Yaskawa INFORM job: test_long_tjr0.JBI

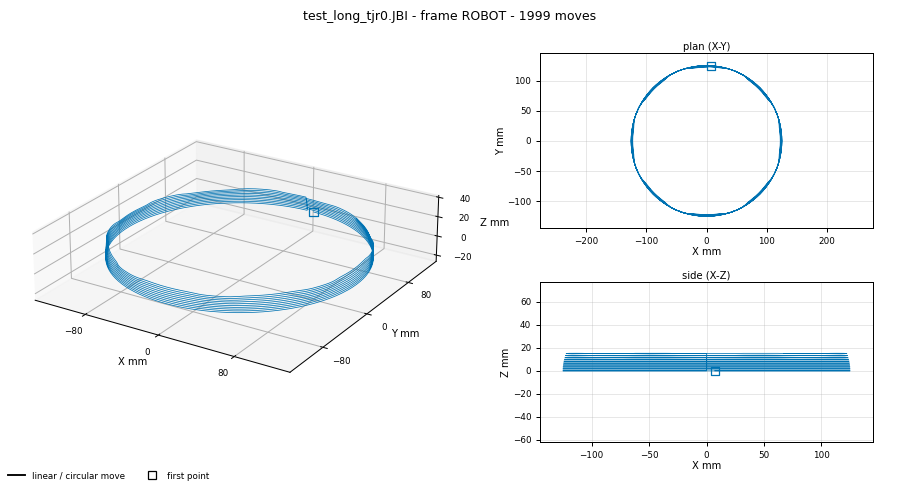
[picture p0: tool path of test_long_tjr0.JBI in frame ROBOT, 1999 of 2000 moves have a stored position in this frame; points joined in program order, loops and branches not executed]
version: 0
/JOB
//NAME test_long
//POS
///NPOS 48,0,0,2,0,0
///TOOL 1
///POSTYPE ROBOT
///RECTAN
///RCONF 1,0,0,0,0,0,0,0,0,0,0,0,0,0,0,0,0,0,0,0,0,0,0,0
C00000=0.000,125.000,0.000,0.0000,0.0000,1.0000
C00001=7.240,124.790,0.000,-0.0000,0.0000,1.0000
C00002=13.740,124.240,0.000,-0.0000,0.0000,1.0000
C00003=19.450,123.480,0.000,-0.0000,0.0000,1.0000
C00004=23.370,122.800,0.000,-0.0000,0.0000,1.0000
C00005=26.070,122.250,0.000,-0.0000,0.0000,1.0000
C00006=28.240,121.770,0.000,-0.0000,-0.0000,1.0000
C00007=30.440,121.240,0.000,-0.0000,-0.0000,1.0000
C00008=33.190,120.510,0.000,-0.0000,0.0000,1.0000
C00009=36.560,119.530,0.000,-0.0000,0.0000,1.0000
C00010=40.120,118.390,0.000,-0.0000,0.0000,1.0000
C00011=43.420,117.220,0.000,-0.0000,0.0000,1.0000
C00012=46.400,116.070,0.000,-0.0000,0.0000,1.0000
C00013=49.260,114.880,0.000,-0.0000,0.0000,1.0000
C00014=52.180,113.590,0.000,-0.0000,0.0000,1.0000
C00015=55.350,112.080,0.000,0.0000,0.0000,1.0000
C00016=58.670,110.370,0.000,0.0000,0.0000,1.0000
C00017=61.750,108.680,0.000,-0.0000,0.0000,1.0000
C00018=64.200,107.250,0.000,-0.0000,0.0000,1.0000
C00019=66.130,106.070,0.000,-0.0000,0.0000,1.0000
C00020=68.010,104.880,0.000,-0.0000,0.0000,1.0000
C00021=70.300,103.360,0.000,-0.0000,0.0000,1.0000
C00022=73.550,101.070,0.000,-0.0000,0.0000,1.0000
C00023=78.140,97.570,0.000,-0.0000,0.0000,1.0000
C00024=83.120,93.360,0.000,-0.0000,0.0000,1.0000
C00025=88.390,88.390,0.000,-0.0000,0.0000,1.0000
C00026=93.360,83.120,0.000,-0.0000,0.0000,1.0000
C00027=97.570,78.140,0.000,-0.0000,0.0000,1.0000
C00028=101.070,73.550,0.000,0.0000,0.0000,1.0000
C00029=103.360,70.300,0.000,-0.0000,0.0000,1.0000
C00030=104.880,68.010,0.000,-0.0000,0.0000,1.0000
C00031=106.070,66.130,0.000,-0.0000,0.0000,1.0000
C00032=107.250,64.200,0.000,-0.0000,0.0000,1.0000
C00033=108.680,61.750,0.000,-0.0000,0.0000,1.0000
C00034=110.370,58.670,0.000,-0.0000,0.0000,1.0000
C00035=112.080,55.350,0.000,-0.0000,0.0000,1.0000
C00036=113.590,52.180,0.000,-0.0000,0.0000,1.0000
C00037=114.880,49.260,0.000,-0.0000,0.0000,1.0000
C00038=116.070,46.400,0.000,-0.0000,0.0000,1.0000
C00039=117.220,43.420,0.000,-0.0000,0.0000,1.0000
C00040=118.390,40.120,0.000,-0.0000,0.0000,1.0000
C00041=119.530,36.560,0.000,-0.0000,0.0000,1.0000
C00042=120.510,33.190,0.000,-0.0000,0.0000,1.0000
C00043=121.240,30.440,0.000,-0.0000,0.0000,1.0000
C00044=121.770,28.240,0.000,-0.0000,0.0000,1.0000
C00045=122.250,26.070,0.000,-0.0000,0.0000,1.0000
C00046=122.800,23.370,0.000,-0.0000,0.0000,1.0000
C00047=123.480,19.450,0.000,-0.0000,0.0000,1.0000
C00048=124.240,13.740,0.000,-0.0000,0.0000,1.0000
C00049=124.790,7.240,0.000,-0.0000,0.0000,1.0000
C00050=125.000,0.000,0.000,-0.0000,0.0000,1.0000
C00051=124.790,-7.240,0.000,0.0000,0.0000,1.0000
C00052=124.240,-13.740,0.000,0.0000,0.0000,1.0000
C00053=123.480,-19.450,0.000,0.0000,0.0000,1.0000
C00054=122.800,-23.370,0.000,0.0000,0.0000,1.0000
C00055=122.250,-26.070,0.000,0.0000,0.0000,1.0000
C00056=121.770,-28.240,0.000,-0.0000,0.0000,1.0000
C00057=121.240,-30.440,0.000,-0.0000,0.0000,1.0000
C00058=120.510,-33.190,0.000,0.0000,0.0000,1.0000
C00059=119.530,-36.560,0.000,0.0000,0.0000,1.0000
C00060=118.390,-40.120,0.000,0.0000,0.0000,1.0000
C00061=117.220,-43.420,0.000,0.0000,0.0000,1.0000
C00062=116.070,-46.400,0.000,0.0000,0.0000,1.0000
C00063=114.880,-49.260,0.000,0.0000,0.0000,1.0000
C00064=113.590,-52.180,0.000,0.0000,0.0000,1.0000
C00065=112.080,-55.350,0.000,0.0000,0.0000,1.0000
C00066=110.370,-58.670,0.000,0.0000,0.0000,1.0000
C00067=108.680,-61.750,0.000,0.0000,0.0000,1.0000
C00068=107.250,-64.200,0.000,0.0000,0.0000,1.0000
C00069=106.070,-66.130,0.000,0.0000,0.0000,1.0000
C00070=104.880,-68.010,0.000,0.0000,0.0000,1.0000
C00071=103.360,-70.300,0.000,0.0000,0.0000,1.0000
C00072=101.070,-73.550,0.000,0.0000,0.0000,1.0000
C00073=97.570,-78.140,0.000,0.0000,0.0000,1.0000
C00074=93.360,-83.120,0.000,0.0000,0.0000,1.0000
C00075=88.390,-88.390,0.000,0.0000,0.0000,1.0000
C00076=83.120,-93.360,0.000,0.0000,0.0000,1.0000
C00077=78.140,-97.570,0.000,0.0000,0.0000,1.0000
C00078=73.550,-101.070,0.000,0.0000,0.0000,1.0000
C00079=70.300,-103.360,0.000,0.0000,0.0000,1.0000
C00080=68.010,-104.880,0.000,0.0000,0.0000,1.0000
C00081=66.130,-106.070,0.000,0.0000,0.0000,1.0000
C00082=64.200,-107.250,0.000,0.0000,0.0000,1.0000
C00083=61.750,-108.680,0.000,0.0000,-0.0000,1.0000
C00084=58.670,-110.370,0.000,0.0000,0.0000,1.0000
C00085=55.350,-112.080,0.000,0.0000,0.0000,1.0000
C00086=52.180,-113.590,0.000,0.0000,0.0000,1.0000
C00087=49.260,-114.880,0.000,0.0000,0.0000,1.0000
C00088=46.400,-116.070,0.000,0.0000,0.0000,1.0000
C00089=43.420,-117.220,0.000,0.0000,0.0000,1.0000
C00090=40.120,-118.390,0.000,0.0000,0.0000,1.0000
C00091=36.560,-119.530,0.000,0.0000,0.0000,1.0000
C00092=33.190,-120.510,0.000,0.0000,0.0000,1.0000
C00093=30.440,-121.240,0.000,0.0000,0.0000,1.0000
C00094=28.240,-121.770,0.000,0.0000,0.0000,1.0000
C00095=26.070,-122.250,0.000,0.0000,0.0000,1.0000
C00096=23.370,-122.800,0.000,0.0000,0.0000,1.0000
C00097=19.450,-123.480,0.000,0.0000,0.0000,1.0000
C00098=13.740,-124.240,0.000,0.0000,0.0000,1.0000
C00099=7.240,-124.790,0.000,0.0000,0.0000,1.0000
C00100=0.000,-125.000,0.000,0.0000,-0.0000,1.0000
C00101=0.000,-125.000,0.000,0.0000,-0.0000,1.0000
C00102=-7.240,-124.790,0.000,0.0000,-0.0000,1.0000
C00103=-13.740,-124.240,0.000,0.0000,-0.0000,1.0000
C00104=-19.450,-123.480,0.000,0.0000,-0.0000,1.0000
C00105=-23.370,-122.800,0.000,-0.0000,-0.0000,1.0000
C00106=-26.070,-122.250,0.000,0.0000,-0.0000,1.0000
C00107=-28.240,-121.770,0.000,0.0000,-0.0000,1.0000
C00108=-30.440,-121.240,0.000,0.0000,-0.0000,1.0000
C00109=-33.190,-120.510,0.000,0.0000,-0.0000,1.0000
C00110=-36.560,-119.530,0.000,0.0000,-0.0000,1.0000
C00111=-40.120,-118.390,0.000,0.0000,-0.0000,1.0000
C00112=-43.420,-117.220,0.000,0.0000,-0.0000,1.0000
C00113=-46.400,-116.070,0.000,0.0000,-0.0000,1.0000
C00114=-49.260,-114.880,0.000,0.0000,-0.0000,1.0000
C00115=-52.180,-113.590,0.000,0.0000,-0.0000,1.0000
C00116=-55.350,-112.080,0.000,0.0000,-0.0000,1.0000
C00117=-58.670,-110.370,0.000,0.0000,-0.0000,1.0000
C00118=-61.750,-108.680,0.000,0.0000,-0.0000,1.0000
C00119=-64.200,-107.250,0.000,0.0000,-0.0000,1.0000
C00120=-66.130,-106.070,0.000,0.0000,-0.0000,1.0000
C00121=-68.010,-104.880,0.000,0.0000,-0.0000,1.0000
C00122=-70.300,-103.360,0.000,0.0000,-0.0000,1.0000
C00123=-73.550,-101.070,0.000,0.0000,-0.0000,1.0000
C00124=-78.140,-97.570,0.000,0.0000,-0.0000,1.0000
C00125=-83.120,-93.360,0.000,0.0000,-0.0000,1.0000
C00126=-88.390,-88.390,0.000,0.0000,-0.0000,1.0000
C00127=-93.360,-83.120,0.000,0.0000,-0.0000,1.0000
C00128=-97.570,-78.140,0.000,0.0000,-0.0000,1.0000
C00129=-101.070,-73.550,0.000,0.0000,-0.0000,1.0000
C00130=-103.360,-70.300,0.000,0.0000,-0.0000,1.0000
C00131=-104.880,-68.010,0.000,0.0000,-0.0000,1.0000
C00132=-106.070,-66.130,0.000,0.0000,-0.0000,1.0000
C00133=-107.250,-64.200,0.000,0.0000,-0.0000,1.0000
C00134=-108.680,-61.750,0.000,0.0000,-0.0000,1.0000
C00135=-110.370,-58.670,0.000,0.0000,-0.0000,1.0000
C00136=-112.080,-55.350,0.000,0.0000,-0.0000,1.0000
C00137=-113.590,-52.180,0.000,0.0000,0.0000,1.0000
C00138=-114.880,-49.260,0.000,0.0000,0.0000,1.0000
C00139=-116.070,-46.400,0.000,0.0000,-0.0000,1.0000
C00140=-117.220,-43.420,0.000,0.0000,-0.0000,1.0000
C00141=-118.390,-40.120,0.000,0.0000,0.0000,1.0000
C00142=-119.530,-36.560,0.000,0.0000,0.0000,1.0000
C00143=-120.510,-33.190,0.000,0.0000,-0.0000,1.0000
C00144=-121.240,-30.440,0.000,0.0000,-0.0000,1.0000
C00145=-121.770,-28.240,0.000,0.0000,-0.0000,1.0000
C00146=-122.250,-26.070,0.000,0.0000,-0.0000,1.0000
C00147=-122.800,-23.370,0.000,0.0000,-0.0000,1.0000
C00148=-123.480,-19.450,0.000,0.0000,-0.0000,1.0000
C00149=-124.240,-13.740,0.000,0.0000,-0.0000,1.0000
C00150=-124.790,-7.240,0.000,0.0000,-0.0000,1.0000
C00151=-125.000,0.000,0.000,0.0000,0.0000,1.0000
C00152=-124.790,7.240,0.000,0.0000,0.0000,1.0000
C00153=-124.240,13.740,0.000,0.0000,0.0000,1.0000
C00154=-123.480,19.450,0.000,0.0000,0.0000,1.0000
C00155=-122.800,23.370,0.000,0.0000,0.0000,1.0000
C00156=-122.250,26.070,0.000,0.0000,0.0000,1.0000
C00157=-121.770,28.240,0.000,0.0000,0.0000,1.0000
C00158=-121.240,30.440,0.000,0.0000,0.0000,1.0000
C00159=-120.510,33.190,0.000,0.0000,0.0000,1.0000
C00160=-119.530,36.560,0.000,0.0000,0.0000,1.0000
C00161=-118.390,40.120,0.000,0.0000,0.0000,1.0000
C00162=-117.220,43.420,0.000,0.0000,0.0000,1.0000
C00163=-116.070,46.400,0.000,0.0000,0.0000,1.0000
C00164=-114.880,49.260,0.000,0.0000,0.0000,1.0000
C00165=-113.590,52.180,0.000,0.0000,0.0000,1.0000
C00166=-112.080,55.350,0.000,0.0000,0.0000,1.0000
C00167=-110.370,58.670,0.000,0.0000,0.0000,1.0000
C00168=-108.680,61.750,0.000,0.0000,0.0000,1.0000
C00169=-107.250,64.200,0.000,0.0000,0.0000,1.0000
C00170=-106.070,66.130,0.000,0.0000,0.0000,1.0000
C00171=-104.880,68.010,0.000,0.0000,0.0000,1.0000
C00172=-103.360,70.300,0.000,0.0000,0.0000,1.0000
C00173=-101.070,73.550,0.000,0.0000,0.0000,1.0000
C00174=-97.570,78.140,0.000,0.0000,0.0000,1.0000
C00175=-93.360,83.120,0.000,0.0000,0.0000,1.0000
C00176=-88.390,88.390,0.000,0.0000,0.0000,1.0000
C00177=-83.120,93.360,0.000,0.0000,0.0000,1.0000
C00178=-78.140,97.570,0.000,0.0000,0.0000,1.0000
C00179=-73.550,101.070,0.000,0.0000,0.0000,1.0000
C00180=-70.300,103.360,0.000,0.0000,0.0000,1.0000
C00181=-68.010,104.880,0.000,0.0000,0.0000,1.0000
C00182=-66.130,106.070,0.000,0.0000,0.0000,1.0000
C00183=-64.200,107.250,0.000,0.0000,0.0000,1.0000
C00184=-61.750,108.680,0.000,0.0000,0.0000,1.0000
C00185=-58.670,110.370,0.000,0.0000,0.0000,1.0000
C00186=-55.350,112.080,0.000,0.0000,0.0000,1.0000
C00187=-52.180,113.590,0.000,0.0000,0.0000,1.0000
C00188=-49.260,114.880,0.000,0.0000,0.0000,1.0000
C00189=-46.400,116.070,0.000,0.0000,0.0000,1.0000
C00190=-43.420,117.220,0.000,0.0000,0.0000,1.0000
C00191=-40.120,118.390,0.000,0.0000,-0.0000,1.0000
C00192=-36.560,119.530,0.000,0.0000,-0.0000,1.0000
C00193=-33.190,120.510,0.000,0.0000,0.0000,1.0000
C00194=-30.440,121.240,0.000,0.0000,0.0000,1.0000
C00195=-28.240,121.770,0.000,0.0000,0.0000,1.0000
C00196=-26.070,122.250,0.000,0.0000,0.0000,1.0000
C00197=-23.370,122.800,0.000,0.0000,0.0000,1.0000
C00198=-19.450,123.480,0.000,0.0000,0.0000,1.0000
C00199=-13.740,124.240,0.000,0.0000,0.0000,1.0000
C00200=-7.240,124.790,0.000,0.0000,0.0000,1.0000
C00201=0.000,125.000,0.000,0.0000,0.0000,1.0000
C00202=0.000,124.960,1.700,0.0000,-0.0400,1.0000
C00203=-7.240,124.750,1.700,0.0000,-0.0400,1.0000
C00204=-13.730,124.210,1.700,0.0000,-0.0400,1.0000
C00205=-19.450,123.440,1.700,0.0100,-0.0400,1.0000
C00206=-23.360,122.760,1.700,0.0100,-0.0400,1.0000
C00207=-26.060,122.230,1.700,0.0100,-0.0300,1.0000
C00208=-28.230,121.750,1.700,0.0100,-0.0200,1.0000
C00209=-30.430,121.230,1.700,0.0000,-0.0200,1.0000
C00210=-33.180,120.510,1.700,0.0000,-0.0100,1.0000
C00211=-36.550,119.530,1.700,0.0000,-0.0000,1.0000
C00212=-40.110,118.390,1.700,0.0000,-0.0000,1.0000
C00213=-43.420,117.220,1.700,0.0000,-0.0000,1.0000
C00214=-46.400,116.070,1.700,0.0000,-0.0000,1.0000
C00215=-49.260,114.880,1.700,0.0000,-0.0000,1.0000
C00216=-52.180,113.590,1.700,0.0000,-0.0000,1.0000
C00217=-55.350,112.080,1.700,0.0000,-0.0000,1.0000
C00218=-58.680,110.370,1.700,0.0000,-0.0000,1.0000
C00219=-61.750,108.670,1.700,0.0100,-0.0100,1.0000
C00220=-64.200,107.240,1.700,0.0100,-0.0100,1.0000
C00221=-66.130,106.050,1.700,0.0100,-0.0200,1.0000
C00222=-68.000,104.850,1.700,0.0200,-0.0300,1.0000
C00223=-70.290,103.330,1.700,0.0200,-0.0300,1.0000
C00224=-73.530,101.040,1.700,0.0300,-0.0300,1.0000
C00225=-78.120,97.540,1.700,0.0300,-0.0300,1.0000
C00226=-83.100,93.330,1.700,0.0300,-0.0300,1.0000
C00227=-88.360,88.360,1.700,0.0300,-0.0300,1.0000
C00228=-93.330,83.100,1.700,0.0300,-0.0300,1.0000
C00229=-97.540,78.120,1.700,0.0300,-0.0300,1.0000
C00230=-101.040,73.530,1.700,0.0300,-0.0300,1.0000
C00231=-103.330,70.290,1.700,0.0300,-0.0200,1.0000
C00232=-104.850,68.000,1.700,0.0300,-0.0200,1.0000
C00233=-106.050,66.130,1.700,0.0200,-0.0100,1.0000
C00234=-107.240,64.200,1.700,0.0100,-0.0100,1.0000
C00235=-108.670,61.750,1.700,0.0100,-0.0100,1.0000
C00236=-110.370,58.680,1.700,0.0000,-0.0000,1.0000
C00237=-112.080,55.350,1.700,0.0000,-0.0000,1.0000
C00238=-113.590,52.180,1.700,0.0000,-0.0000,1.0000
C00239=-114.880,49.260,1.700,0.0000,-0.0000,1.0000
C00240=-116.070,46.400,1.700,0.0000,-0.0000,1.0000
C00241=-117.220,43.420,1.700,0.0000,-0.0000,1.0000
C00242=-118.390,40.110,1.700,0.0000,-0.0000,1.0000
C00243=-119.530,36.550,1.700,0.0000,-0.0000,1.0000
C00244=-120.510,33.180,1.700,0.0100,-0.0000,1.0000
C00245=-121.230,30.430,1.700,0.0200,-0.0000,1.0000
C00246=-121.750,28.230,1.700,0.0200,-0.0100,1.0000
C00247=-122.230,26.060,1.700,0.0300,-0.0100,1.0000
C00248=-122.760,23.360,1.700,0.0400,-0.0100,1.0000
C00249=-123.440,19.450,1.700,0.0400,-0.0100,1.0000
C00250=-124.210,13.730,1.700,0.0400,-0.0000,1.0000
C00251=-124.750,7.240,1.700,0.0400,-0.0000,1.0000
C00252=-124.960,0.000,1.700,0.0400,-0.0000,1.0000
C00253=-124.750,-7.240,1.700,0.0400,0.0000,1.0000
C00254=-124.210,-13.730,1.700,0.0400,0.0000,1.0000
C00255=-123.440,-19.450,1.700,0.0400,0.0100,1.0000
C00256=-122.760,-23.360,1.700,0.0400,0.0100,1.0000
C00257=-122.230,-26.060,1.700,0.0300,0.0100,1.0000
C00258=-121.750,-28.230,1.700,0.0200,0.0100,1.0000
C00259=-121.230,-30.430,1.700,0.0200,0.0000,1.0000
C00260=-120.510,-33.180,1.700,0.0100,0.0000,1.0000
C00261=-119.530,-36.550,1.700,0.0000,0.0000,1.0000
C00262=-118.390,-40.110,1.700,0.0000,0.0000,1.0000
C00263=-117.220,-43.420,1.700,0.0000,0.0000,1.0000
C00264=-116.070,-46.400,1.700,0.0000,0.0000,1.0000
C00265=-114.880,-49.260,1.700,0.0000,0.0000,1.0000
C00266=-113.590,-52.180,1.700,0.0000,0.0000,1.0000
C00267=-112.080,-55.350,1.700,0.0000,0.0000,1.0000
C00268=-110.370,-58.680,1.700,0.0000,0.0000,1.0000
C00269=-108.670,-61.750,1.700,0.0100,0.0100,1.0000
C00270=-107.240,-64.200,1.700,0.0100,0.0100,1.0000
C00271=-106.050,-66.130,1.700,0.0200,0.0100,1.0000
C00272=-104.850,-68.000,1.700,0.0300,0.0200,1.0000
C00273=-103.330,-70.290,1.700,0.0300,0.0200,1.0000
C00274=-101.040,-73.530,1.700,0.0300,0.0300,1.0000
C00275=-97.540,-78.120,1.700,0.0300,0.0300,1.0000
C00276=-93.330,-83.100,1.700,0.0300,0.0300,1.0000
C00277=-88.360,-88.360,1.700,0.0300,0.0300,1.0000
C00278=-83.100,-93.330,1.700,0.0300,0.0300,1.0000
C00279=-78.120,-97.540,1.700,0.0300,0.0300,1.0000
C00280=-73.530,-101.040,1.700,0.0300,0.0300,1.0000
C00281=-70.290,-103.330,1.700,0.0200,0.0300,1.0000
C00282=-68.000,-104.850,1.700,0.0200,0.0300,1.0000
C00283=-66.130,-106.050,1.700,0.0100,0.0200,1.0000
C00284=-64.200,-107.240,1.700,0.0100,0.0100,1.0000
C00285=-61.750,-108.670,1.700,0.0100,0.0100,1.0000
C00286=-58.680,-110.370,1.700,0.0000,0.0000,1.0000
C00287=-55.350,-112.080,1.700,0.0000,0.0000,1.0000
C00288=-52.180,-113.590,1.700,0.0000,0.0000,1.0000
C00289=-49.260,-114.880,1.700,0.0000,0.0000,1.0000
C00290=-46.400,-116.070,1.700,0.0000,0.0000,1.0000
C00291=-43.420,-117.220,1.700,0.0000,0.0000,1.0000
C00292=-40.110,-118.390,1.700,0.0000,0.0000,1.0000
C00293=-36.550,-119.530,1.700,0.0000,0.0000,1.0000
C00294=-33.180,-120.510,1.700,0.0000,0.0100,1.0000
C00295=-30.430,-121.230,1.700,0.0000,0.0200,1.0000
C00296=-28.230,-121.750,1.700,0.0100,0.0200,1.0000
C00297=-26.060,-122.230,1.700,0.0100,0.0300,1.0000
C00298=-23.360,-122.760,1.700,0.0100,0.0400,1.0000
C00299=-19.450,-123.440,1.700,0.0100,0.0400,1.0000
C00300=-13.730,-124.210,1.700,0.0000,0.0400,1.0000
C00301=-7.240,-124.750,1.700,0.0000,0.0400,1.0000
C00302=0.000,-124.960,1.700,0.0000,0.0400,1.0000
C00303=0.000,-124.960,1.700,0.0000,0.0400,1.0000
C00304=7.240,-124.750,1.700,-0.0000,0.0400,1.0000
C00305=13.730,-124.210,1.700,-0.0000,0.0400,1.0000
C00306=19.450,-123.440,1.700,-0.0100,0.0400,1.0000
C00307=23.360,-122.760,1.700,-0.0100,0.0400,1.0000
C00308=26.060,-122.230,1.700,-0.0100,0.0300,1.0000
C00309=28.230,-121.750,1.700,-0.0100,0.0200,1.0000
C00310=30.430,-121.230,1.700,-0.0000,0.0200,1.0000
C00311=33.180,-120.510,1.700,-0.0000,0.0100,1.0000
C00312=36.550,-119.530,1.700,-0.0000,0.0000,1.0000
C00313=40.110,-118.390,1.700,-0.0000,0.0000,1.0000
C00314=43.420,-117.220,1.700,-0.0000,0.0000,1.0000
C00315=46.400,-116.070,1.700,-0.0000,0.0000,1.0000
C00316=49.260,-114.880,1.700,-0.0000,0.0000,1.0000
C00317=52.180,-113.590,1.700,-0.0000,0.0000,1.0000
C00318=55.350,-112.080,1.700,-0.0000,0.0000,1.0000
C00319=58.680,-110.370,1.700,-0.0000,0.0000,1.0000
C00320=61.750,-108.670,1.700,-0.0100,0.0100,1.0000
C00321=64.200,-107.240,1.700,-0.0100,0.0100,1.0000
C00322=66.130,-106.050,1.700,-0.0100,0.0200,1.0000
C00323=68.000,-104.850,1.700,-0.0200,0.0300,1.0000
C00324=70.290,-103.330,1.700,-0.0200,0.0300,1.0000
C00325=73.530,-101.040,1.700,-0.0300,0.0300,1.0000
C00326=78.120,-97.540,1.700,-0.0300,0.0300,1.0000
C00327=83.100,-93.330,1.700,-0.0300,0.0300,1.0000
C00328=88.360,-88.360,1.700,-0.0300,0.0300,1.0000
C00329=93.330,-83.100,1.700,-0.0300,0.0300,1.0000
C00330=97.540,-78.120,1.700,-0.0300,0.0300,1.0000
C00331=101.040,-73.530,1.700,-0.0300,0.0300,1.0000
C00332=103.330,-70.290,1.700,-0.0300,0.0200,1.0000
C00333=104.850,-68.000,1.700,-0.0300,0.0200,1.0000
C00334=106.050,-66.130,1.700,-0.0200,0.0100,1.0000
C00335=107.240,-64.200,1.700,-0.0100,0.0100,1.0000
C00336=108.670,-61.750,1.700,-0.0100,0.0100,1.0000
C00337=110.370,-58.680,1.700,-0.0000,0.0000,1.0000
C00338=112.080,-55.350,1.700,-0.0000,0.0000,1.0000
C00339=113.590,-52.180,1.700,-0.0000,0.0000,1.0000
C00340=114.880,-49.260,1.700,-0.0000,0.0000,1.0000
C00341=116.070,-46.400,1.700,-0.0000,0.0000,1.0000
C00342=117.220,-43.420,1.700,-0.0000,0.0000,1.0000
C00343=118.390,-40.110,1.700,-0.0000,0.0000,1.0000
C00344=119.530,-36.550,1.700,-0.0000,0.0000,1.0000
C00345=120.510,-33.180,1.700,-0.0100,0.0000,1.0000
C00346=121.230,-30.430,1.700,-0.0200,0.0000,1.0000
C00347=121.750,-28.230,1.700,-0.0200,0.0100,1.0000
C00348=122.230,-26.060,1.700,-0.0300,0.0100,1.0000
C00349=122.760,-23.360,1.700,-0.0400,0.0100,1.0000
C00350=123.440,-19.450,1.700,-0.0400,0.0100,1.0000
C00351=124.210,-13.730,1.700,-0.0400,0.0000,1.0000
C00352=124.750,-7.240,1.700,-0.0400,0.0000,1.0000
C00353=124.960,0.000,1.700,-0.0400,0.0000,1.0000
C00354=124.750,7.240,1.700,-0.0400,-0.0000,1.0000
C00355=124.210,13.730,1.700,-0.0400,-0.0000,1.0000
C00356=123.440,19.450,1.700,-0.0400,-0.0100,1.0000
C00357=122.760,23.360,1.700,-0.0400,-0.0100,1.0000
C00358=122.230,26.060,1.700,-0.0300,-0.0100,1.0000
C00359=121.750,28.230,1.700,-0.0200,-0.0100,1.0000
C00360=121.230,30.430,1.700,-0.0200,-0.0000,1.0000
C00361=120.510,33.180,1.700,-0.0100,-0.0000,1.0000
C00362=119.530,36.550,1.700,-0.0000,-0.0000,1.0000
C00363=118.390,40.110,1.700,-0.0000,-0.0000,1.0000
C00364=117.220,43.420,1.700,-0.0000,-0.0000,1.0000
C00365=116.070,46.400,1.700,-0.0000,-0.0000,1.0000
C00366=114.880,49.260,1.700,-0.0000,-0.0000,1.0000
C00367=113.590,52.180,1.700,-0.0000,-0.0000,1.0000
C00368=112.080,55.350,1.700,-0.0000,-0.0000,1.0000
C00369=110.370,58.680,1.700,-0.0000,-0.0000,1.0000
C00370=108.670,61.750,1.700,-0.0100,-0.0100,1.0000
C00371=107.240,64.200,1.700,-0.0100,-0.0100,1.0000
C00372=106.050,66.130,1.700,-0.0200,-0.0100,1.0000
C00373=104.850,68.000,1.700,-0.0300,-0.0200,1.0000
C00374=103.330,70.290,1.700,-0.0300,-0.0200,1.0000
C00375=101.040,73.530,1.700,-0.0300,-0.0300,1.0000
C00376=97.540,78.120,1.700,-0.0300,-0.0300,1.0000
C00377=93.330,83.100,1.700,-0.0300,-0.0300,1.0000
C00378=88.360,88.360,1.700,-0.0300,-0.0300,1.0000
C00379=83.100,93.330,1.700,-0.0300,-0.0300,1.0000
C00380=78.120,97.540,1.700,-0.0300,-0.0300,1.0000
C00381=73.530,101.040,1.700,-0.0300,-0.0300,1.0000
C00382=70.290,103.330,1.700,-0.0200,-0.0300,1.0000
C00383=68.000,104.850,1.700,-0.0200,-0.0300,1.0000
C00384=66.130,106.050,1.700,-0.0100,-0.0200,1.0000
C00385=64.200,107.240,1.700,-0.0100,-0.0100,1.0000
C00386=61.750,108.670,1.700,-0.0100,-0.0100,1.0000
C00387=58.680,110.370,1.700,-0.0000,-0.0000,1.0000
C00388=55.350,112.080,1.700,-0.0000,-0.0000,1.0000
C00389=52.180,113.590,1.700,-0.0000,-0.0000,1.0000
C00390=49.260,114.880,1.700,-0.0000,-0.0000,1.0000
C00391=46.400,116.070,1.700,-0.0000,-0.0000,1.0000
C00392=43.420,117.220,1.700,-0.0000,-0.0000,1.0000
C00393=40.110,118.390,1.700,-0.0000,-0.0000,1.0000
C00394=36.550,119.530,1.700,-0.0000,-0.0000,1.0000
C00395=33.180,120.510,1.700,-0.0000,-0.0100,1.0000
C00396=30.430,121.230,1.700,-0.0000,-0.0200,1.0000
C00397=28.230,121.750,1.700,-0.0100,-0.0200,1.0000
C00398=26.060,122.230,1.700,-0.0100,-0.0300,1.0000
C00399=23.360,122.760,1.700,-0.0100,-0.0400,1.0000
C00400=19.450,123.440,1.700,-0.0100,-0.0400,1.0000
C00401=13.730,124.210,1.700,-0.0000,-0.0400,1.0000
C00402=7.240,124.750,1.700,-0.0000,-0.0400,1.0000
C00403=0.000,124.960,1.700,0.0000,-0.0400,1.0000
C00404=0.000,124.850,3.400,0.0000,-0.0900,1.0000
C00405=7.230,124.640,3.400,-0.0100,-0.0900,1.0000
C00406=13.710,124.100,3.400,-0.0100,-0.0900,1.0000
C00407=19.430,123.340,3.400,-0.0100,-0.0800,1.0000
C00408=23.340,122.670,3.400,-0.0100,-0.0700,1.0000
C00409=26.030,122.150,3.400,-0.0100,-0.0600,1.0000
C00410=28.200,121.690,3.400,-0.0100,-0.0500,1.0000
C00411=30.400,121.190,3.400,-0.0100,-0.0300,1.0000
C00412=33.140,120.490,3.400,-0.0100,-0.0200,1.0000
C00413=36.520,119.530,3.400,-0.0000,-0.0100,1.0000
C00414=40.090,118.390,3.400,-0.0000,-0.0000,1.0000
C00415=43.400,117.220,3.400,-0.0000,-0.0000,1.0000
C00416=46.390,116.070,3.400,-0.0000,-0.0000,1.0000
C00417=49.270,114.880,3.400,-0.0000,-0.0000,1.0000
C00418=52.200,113.580,3.400,-0.0000,-0.0000,1.0000
C00419=55.370,112.060,3.400,-0.0000,-0.0000,1.0000
C00420=58.700,110.340,3.400,-0.0000,-0.0100,1.0000
C00421=61.760,108.640,3.400,-0.0100,-0.0200,1.0000
C00422=64.200,107.190,3.400,-0.0200,-0.0300,1.0000
C00423=66.110,105.990,3.400,-0.0300,-0.0400,1.0000
C00424=67.970,104.780,3.400,-0.0300,-0.0500,1.0000
C00425=70.240,103.240,3.400,-0.0400,-0.0600,1.0000
C00426=73.470,100.950,3.400,-0.0500,-0.0700,1.0000
C00427=78.050,97.450,3.400,-0.0500,-0.0700,1.0000
C00428=83.020,93.240,3.400,-0.0600,-0.0600,1.0000
C00429=88.280,88.280,3.400,-0.0600,-0.0600,1.0000
C00430=93.240,83.020,3.400,-0.0600,-0.0600,1.0000
C00431=97.450,78.050,3.400,-0.0700,-0.0500,1.0000
C00432=100.950,73.470,3.400,-0.0700,-0.0500,1.0000
C00433=103.240,70.240,3.400,-0.0600,-0.0400,1.0000
C00434=104.780,67.970,3.400,-0.0500,-0.0300,1.0000
C00435=105.990,66.110,3.400,-0.0400,-0.0300,1.0000
C00436=107.190,64.200,3.400,-0.0300,-0.0200,1.0000
C00437=108.640,61.760,3.400,-0.0200,-0.0100,1.0000
C00438=110.340,58.700,3.400,-0.0100,-0.0000,1.0000
C00439=112.060,55.370,3.400,-0.0000,-0.0000,1.0000
C00440=113.580,52.200,3.400,-0.0000,-0.0000,1.0000
C00441=114.880,49.270,3.400,-0.0000,-0.0000,1.0000
C00442=116.070,46.390,3.400,-0.0000,-0.0000,1.0000
C00443=117.220,43.400,3.400,-0.0000,-0.0000,1.0000
C00444=118.390,40.090,3.400,-0.0000,-0.0000,1.0000
C00445=119.530,36.520,3.400,-0.0100,-0.0000,1.0000
C00446=120.490,33.140,3.400,-0.0200,-0.0100,1.0000
C00447=121.190,30.400,3.400,-0.0300,-0.0100,1.0000
C00448=121.690,28.200,3.400,-0.0500,-0.0100,1.0000
C00449=122.150,26.030,3.400,-0.0600,-0.0100,1.0000
C00450=122.670,23.340,3.400,-0.0700,-0.0100,1.0000
C00451=123.340,19.430,3.400,-0.0800,-0.0100,1.0000
C00452=124.100,13.710,3.400,-0.0900,-0.0100,1.0000
C00453=124.640,7.230,3.400,-0.0900,-0.0100,1.0000
C00454=124.850,0.000,3.400,-0.0900,0.0000,1.0000
C00455=124.640,-7.230,3.400,-0.0900,0.0100,1.0000
C00456=124.100,-13.710,3.400,-0.0900,0.0100,1.0000
C00457=123.340,-19.430,3.400,-0.0800,0.0100,1.0000
C00458=122.670,-23.340,3.400,-0.0700,0.0100,1.0000
C00459=122.150,-26.030,3.400,-0.0600,0.0100,1.0000
C00460=121.690,-28.200,3.400,-0.0500,0.0100,1.0000
C00461=121.190,-30.400,3.400,-0.0300,0.0100,1.0000
C00462=120.490,-33.140,3.400,-0.0200,0.0100,1.0000
C00463=119.530,-36.520,3.400,-0.0100,0.0000,1.0000
C00464=118.390,-40.090,3.400,-0.0000,0.0000,1.0000
C00465=117.220,-43.400,3.400,-0.0000,0.0000,1.0000
C00466=116.070,-46.390,3.400,-0.0000,0.0000,1.0000
C00467=114.880,-49.270,3.400,-0.0000,0.0000,1.0000
C00468=113.580,-52.200,3.400,-0.0000,0.0000,1.0000
C00469=112.060,-55.370,3.400,-0.0000,0.0000,1.0000
C00470=110.340,-58.700,3.400,-0.0100,0.0000,1.0000
C00471=108.640,-61.760,3.400,-0.0200,0.0100,1.0000
C00472=107.190,-64.200,3.400,-0.0300,0.0200,1.0000
C00473=105.990,-66.110,3.400,-0.0400,0.0300,1.0000
C00474=104.780,-67.970,3.400,-0.0500,0.0300,1.0000
C00475=103.240,-70.240,3.400,-0.0600,0.0400,1.0000
C00476=100.950,-73.470,3.400,-0.0700,0.0500,1.0000
C00477=97.450,-78.050,3.400,-0.0700,0.0500,1.0000
C00478=93.240,-83.020,3.400,-0.0600,0.0600,1.0000
C00479=88.280,-88.280,3.400,-0.0600,0.0600,1.0000
C00480=83.020,-93.240,3.400,-0.0600,0.0600,1.0000
C00481=78.050,-97.450,3.400,-0.0500,0.0700,1.0000
C00482=73.470,-100.950,3.400,-0.0500,0.0700,1.0000
C00483=70.240,-103.240,3.400,-0.0400,0.0600,1.0000
C00484=67.970,-104.780,3.400,-0.0300,0.0500,1.0000
C00485=66.110,-105.990,3.400,-0.0300,0.0400,1.0000
C00486=64.200,-107.190,3.400,-0.0200,0.0300,1.0000
C00487=61.760,-108.640,3.400,-0.0100,0.0200,1.0000
C00488=58.700,-110.340,3.400,-0.0000,0.0100,1.0000
C00489=55.370,-112.060,3.400,-0.0000,0.0000,1.0000
C00490=52.200,-113.580,3.400,-0.0000,0.0000,1.0000
C00491=49.270,-114.880,3.400,-0.0000,0.0000,1.0000
C00492=46.390,-116.070,3.400,-0.0000,0.0000,1.0000
C00493=43.400,-117.220,3.400,-0.0000,0.0000,1.0000
C00494=40.090,-118.390,3.400,-0.0000,0.0000,1.0000
C00495=36.520,-119.530,3.400,-0.0000,0.0100,1.0000
C00496=33.140,-120.490,3.400,-0.0100,0.0200,1.0000
C00497=30.400,-121.190,3.400,-0.0100,0.0300,1.0000
C00498=28.200,-121.690,3.400,-0.0100,0.0500,1.0000
C00499=26.030,-122.150,3.400,-0.0100,0.0600,1.0000
C00500=23.340,-122.670,3.400,-0.0100,0.0700,1.0000
C00501=19.430,-123.340,3.400,-0.0100,0.0800,1.0000
C00502=13.710,-124.100,3.400,-0.0100,0.0900,1.0000
C00503=7.230,-124.640,3.400,-0.0100,0.0900,1.0000
C00504=0.000,-124.850,3.400,0.0000,0.0900,1.0000
C00505=0.000,-124.850,3.400,0.0000,0.0900,1.0000
C00506=-7.230,-124.640,3.400,0.0100,0.0900,1.0000
C00507=-13.710,-124.100,3.400,0.0100,0.0900,1.0000
C00508=-19.430,-123.340,3.400,0.0100,0.0800,1.0000
C00509=-23.340,-122.670,3.400,0.0100,0.0700,1.0000
C00510=-26.030,-122.150,3.400,0.0100,0.0600,1.0000
C00511=-28.200,-121.690,3.400,0.0100,0.0500,1.0000
C00512=-30.400,-121.190,3.400,0.0100,0.0300,1.0000
C00513=-33.140,-120.490,3.400,0.0100,0.0200,1.0000
C00514=-36.520,-119.530,3.400,0.0000,0.0100,1.0000
C00515=-40.090,-118.390,3.400,0.0000,0.0000,1.0000
C00516=-43.400,-117.220,3.400,0.0000,0.0000,1.0000
C00517=-46.390,-116.070,3.400,0.0000,0.0000,1.0000
C00518=-49.270,-114.880,3.400,0.0000,0.0000,1.0000
C00519=-52.200,-113.580,3.400,0.0000,0.0000,1.0000
C00520=-55.370,-112.060,3.400,0.0000,0.0000,1.0000
C00521=-58.700,-110.340,3.400,0.0000,0.0100,1.0000
C00522=-61.760,-108.640,3.400,0.0100,0.0200,1.0000
C00523=-64.200,-107.190,3.400,0.0200,0.0300,1.0000
C00524=-66.110,-105.990,3.400,0.0300,0.0400,1.0000
C00525=-67.970,-104.780,3.400,0.0300,0.0500,1.0000
C00526=-70.240,-103.240,3.400,0.0400,0.0600,1.0000
C00527=-73.470,-100.950,3.400,0.0500,0.0700,1.0000
C00528=-78.050,-97.450,3.400,0.0500,0.0700,1.0000
C00529=-83.020,-93.240,3.400,0.0600,0.0600,1.0000
C00530=-88.280,-88.280,3.400,0.0600,0.0600,1.0000
C00531=-93.240,-83.020,3.400,0.0600,0.0600,1.0000
C00532=-97.450,-78.050,3.400,0.0700,0.0500,1.0000
C00533=-100.950,-73.470,3.400,0.0700,0.0500,1.0000
C00534=-103.240,-70.240,3.400,0.0600,0.0400,1.0000
C00535=-104.780,-67.970,3.400,0.0500,0.0300,1.0000
C00536=-105.990,-66.110,3.400,0.0400,0.0300,1.0000
C00537=-107.190,-64.200,3.400,0.0300,0.0200,1.0000
C00538=-108.640,-61.760,3.400,0.0200,0.0100,1.0000
C00539=-110.340,-58.700,3.400,0.0100,0.0000,1.0000
C00540=-112.060,-55.370,3.400,0.0000,0.0000,1.0000
C00541=-113.580,-52.200,3.400,0.0000,0.0000,1.0000
C00542=-114.880,-49.270,3.400,0.0000,0.0000,1.0000
C00543=-116.070,-46.390,3.400,0.0000,0.0000,1.0000
C00544=-117.220,-43.400,3.400,0.0000,0.0000,1.0000
C00545=-118.390,-40.090,3.400,0.0000,0.0000,1.0000
C00546=-119.530,-36.520,3.400,0.0100,0.0000,1.0000
C00547=-120.490,-33.140,3.400,0.0200,0.0100,1.0000
C00548=-121.190,-30.400,3.400,0.0300,0.0100,1.0000
C00549=-121.690,-28.200,3.400,0.0500,0.0100,1.0000
C00550=-122.150,-26.030,3.400,0.0600,0.0100,1.0000
C00551=-122.670,-23.340,3.400,0.0700,0.0100,1.0000
C00552=-123.340,-19.430,3.400,0.0800,0.0100,1.0000
C00553=-124.100,-13.710,3.400,0.0900,0.0100,1.0000
C00554=-124.640,-7.230,3.400,0.0900,0.0100,1.0000
C00555=-124.850,0.000,3.400,0.0900,-0.0000,1.0000
C00556=-124.640,7.230,3.400,0.0900,-0.0100,1.0000
C00557=-124.100,13.710,3.400,0.0900,-0.0100,1.0000
C00558=-123.340,19.430,3.400,0.0800,-0.0100,1.0000
C00559=-122.670,23.340,3.400,0.0700,-0.0100,1.0000
C00560=-122.150,26.030,3.400,0.0600,-0.0100,1.0000
C00561=-121.690,28.200,3.400,0.0500,-0.0100,1.0000
C00562=-121.190,30.400,3.400,0.0300,-0.0100,1.0000
C00563=-120.490,33.140,3.400,0.0200,-0.0100,1.0000
C00564=-119.530,36.520,3.400,0.0100,-0.0000,1.0000
C00565=-118.390,40.090,3.400,0.0000,-0.0000,1.0000
C00566=-117.220,43.400,3.400,0.0000,-0.0000,1.0000
C00567=-116.070,46.390,3.400,0.0000,-0.0000,1.0000
C00568=-114.880,49.270,3.400,0.0000,-0.0000,1.0000
C00569=-113.580,52.200,3.400,0.0000,-0.0000,1.0000
C00570=-112.060,55.370,3.400,0.0000,-0.0000,1.0000
C00571=-110.340,58.700,3.400,0.0100,-0.0000,1.0000
C00572=-108.640,61.760,3.400,0.0200,-0.0100,1.0000
C00573=-107.190,64.200,3.400,0.0300,-0.0200,1.0000
C00574=-105.990,66.110,3.400,0.0400,-0.0300,1.0000
C00575=-104.780,67.970,3.400,0.0500,-0.0300,1.0000
C00576=-103.240,70.240,3.400,0.0600,-0.0400,1.0000
C00577=-100.950,73.470,3.400,0.0700,-0.0500,1.0000
C00578=-97.450,78.050,3.400,0.0700,-0.0500,1.0000
C00579=-93.240,83.020,3.400,0.0600,-0.0600,1.0000
C00580=-88.280,88.280,3.400,0.0600,-0.0600,1.0000
C00581=-83.020,93.240,3.400,0.0600,-0.0600,1.0000
C00582=-78.050,97.450,3.400,0.0500,-0.0700,1.0000
C00583=-73.470,100.950,3.400,0.0500,-0.0700,1.0000
C00584=-70.240,103.240,3.400,0.0400,-0.0600,1.0000
C00585=-67.970,104.780,3.400,0.0300,-0.0500,1.0000
C00586=-66.110,105.990,3.400,0.0300,-0.0400,1.0000
C00587=-64.200,107.190,3.400,0.0200,-0.0300,1.0000
C00588=-61.760,108.640,3.400,0.0100,-0.0200,1.0000
C00589=-58.700,110.340,3.400,0.0000,-0.0100,1.0000
C00590=-55.370,112.060,3.400,0.0000,-0.0000,1.0000
C00591=-52.200,113.580,3.400,0.0000,-0.0000,1.0000
C00592=-49.270,114.880,3.400,0.0000,-0.0000,1.0000
C00593=-46.390,116.070,3.400,0.0000,-0.0000,1.0000
C00594=-43.400,117.220,3.400,0.0000,-0.0000,1.0000
C00595=-40.090,118.390,3.400,0.0000,-0.0000,1.0000
C00596=-36.520,119.530,3.400,0.0000,-0.0100,1.0000
C00597=-33.140,120.490,3.400,0.0100,-0.0200,1.0000
C00598=-30.400,121.190,3.400,0.0100,-0.0300,1.0000
C00599=-28.200,121.690,3.400,0.0100,-0.0500,1.0000
C00600=-26.030,122.150,3.400,0.0100,-0.0600,1.0000
C00601=-23.340,122.670,3.400,0.0100,-0.0700,1.0000
C00602=-19.430,123.340,3.400,0.0100,-0.0800,1.0000
C00603=-13.710,124.100,3.400,0.0100,-0.0900,1.0000
C00604=-7.230,124.640,3.400,0.0100,-0.0900,1.0000
C00605=0.000,124.850,3.400,0.0000,-0.0900,1.0000
C00606=0.000,124.670,5.090,0.0000,-0.1300,0.9900
C00607=-7.210,124.460,5.090,0.0100,-0.1300,0.9900
C00608=-13.680,123.910,5.090,0.0100,-0.1300,0.9900
C00609=-19.390,123.160,5.090,0.0200,-0.1200,0.9900
C00610=-23.300,122.520,5.090,0.0200,-0.1100,0.9900
C00611=-25.990,122.020,5.090,0.0200,-0.0900,1.0000
C00612=-28.160,121.600,5.100,0.0100,-0.0700,1.0000
C00613=-30.350,121.130,5.100,0.0100,-0.0500,1.0000
C00614=-33.090,120.460,5.100,0.0100,-0.0300,1.0000
C00615=-36.470,119.520,5.100,0.0000,-0.0100,1.0000
C00616=-40.050,118.400,5.100,0.0000,-0.0000,1.0000
C00617=-43.380,117.230,5.100,0.0000,-0.0000,1.0000
C00618=-46.390,116.070,5.100,0.0000,-0.0000,1.0000
C00619=-49.280,114.880,5.100,0.0000,-0.0000,1.0000
C00620=-52.220,113.570,5.100,0.0000,-0.0000,1.0000
C00621=-55.410,112.040,5.100,0.0000,-0.0000,1.0000
C00622=-58.730,110.300,5.100,0.0100,-0.0100,1.0000
C00623=-61.780,108.580,5.100,0.0100,-0.0300,1.0000
C00624=-64.190,107.110,5.100,0.0300,-0.0400,1.0000
C00625=-66.080,105.890,5.100,0.0400,-0.0600,1.0000
C00626=-67.910,104.660,5.090,0.0500,-0.0800,1.0000
C00627=-70.160,103.110,5.090,0.0600,-0.0900,0.9900
C00628=-73.380,100.800,5.090,0.0700,-0.1000,0.9900
C00629=-77.940,97.300,5.090,0.0800,-0.1000,0.9900
C00630=-82.910,93.100,5.090,0.0900,-0.1000,0.9900
C00631=-88.150,88.150,5.090,0.0900,-0.0900,0.9900
C00632=-93.100,82.910,5.090,0.1000,-0.0900,0.9900
C00633=-97.300,77.940,5.090,0.1000,-0.0800,0.9900
C00634=-100.800,73.380,5.090,0.1000,-0.0700,0.9900
C00635=-103.110,70.160,5.090,0.0900,-0.0600,0.9900
C00636=-104.660,67.910,5.090,0.0800,-0.0500,1.0000
C00637=-105.890,66.080,5.100,0.0600,-0.0400,1.0000
C00638=-107.110,64.190,5.100,0.0400,-0.0300,1.0000
C00639=-108.580,61.780,5.100,0.0300,-0.0100,1.0000
C00640=-110.300,58.730,5.100,0.0100,-0.0100,1.0000
C00641=-112.040,55.410,5.100,0.0000,-0.0000,1.0000
C00642=-113.570,52.220,5.100,0.0000,-0.0000,1.0000
C00643=-114.880,49.280,5.100,0.0000,-0.0000,1.0000
C00644=-116.070,46.390,5.100,0.0000,-0.0000,1.0000
C00645=-117.230,43.380,5.100,0.0000,-0.0000,1.0000
C00646=-118.400,40.050,5.100,0.0000,-0.0000,1.0000
C00647=-119.520,36.470,5.100,0.0100,-0.0000,1.0000
C00648=-120.460,33.090,5.100,0.0300,-0.0100,1.0000
C00649=-121.130,30.350,5.100,0.0500,-0.0100,1.0000
C00650=-121.600,28.160,5.100,0.0700,-0.0100,1.0000
C00651=-122.020,25.990,5.090,0.0900,-0.0200,1.0000
C00652=-122.520,23.300,5.090,0.1100,-0.0200,0.9900
C00653=-123.160,19.390,5.090,0.1200,-0.0200,0.9900
C00654=-123.910,13.680,5.090,0.1300,-0.0100,0.9900
C00655=-124.460,7.210,5.090,0.1300,-0.0100,0.9900
C00656=-124.670,0.000,5.090,0.1300,-0.0000,0.9900
C00657=-124.460,-7.210,5.090,0.1300,0.0100,0.9900
C00658=-123.910,-13.680,5.090,0.1300,0.0100,0.9900
C00659=-123.160,-19.390,5.090,0.1200,0.0200,0.9900
C00660=-122.520,-23.300,5.090,0.1100,0.0200,0.9900
C00661=-122.020,-25.990,5.090,0.0900,0.0200,1.0000
C00662=-121.600,-28.160,5.100,0.0700,0.0100,1.0000
C00663=-121.130,-30.350,5.100,0.0500,0.0100,1.0000
C00664=-120.460,-33.090,5.100,0.0300,0.0100,1.0000
C00665=-119.520,-36.470,5.100,0.0100,0.0000,1.0000
C00666=-118.400,-40.050,5.100,0.0000,0.0000,1.0000
C00667=-117.230,-43.380,5.100,0.0000,0.0000,1.0000
C00668=-116.070,-46.390,5.100,0.0000,0.0000,1.0000
C00669=-114.880,-49.280,5.100,0.0000,0.0000,1.0000
C00670=-113.570,-52.220,5.100,0.0000,0.0000,1.0000
C00671=-112.040,-55.410,5.100,0.0000,0.0000,1.0000
C00672=-110.300,-58.730,5.100,0.0100,0.0100,1.0000
C00673=-108.580,-61.780,5.100,0.0300,0.0100,1.0000
C00674=-107.110,-64.190,5.100,0.0400,0.0300,1.0000
C00675=-105.890,-66.080,5.100,0.0600,0.0400,1.0000
C00676=-104.660,-67.910,5.090,0.0800,0.0500,1.0000
C00677=-103.110,-70.160,5.090,0.0900,0.0600,0.9900
C00678=-100.800,-73.380,5.090,0.1000,0.0700,0.9900
C00679=-97.300,-77.940,5.090,0.1000,0.0800,0.9900
C00680=-93.100,-82.910,5.090,0.1000,0.0900,0.9900
C00681=-88.150,-88.150,5.090,0.0900,0.0900,0.9900
C00682=-82.910,-93.100,5.090,0.0900,0.1000,0.9900
C00683=-77.940,-97.300,5.090,0.0800,0.1000,0.9900
C00684=-73.380,-100.800,5.090,0.0700,0.1000,0.9900
C00685=-70.160,-103.110,5.090,0.0600,0.0900,0.9900
C00686=-67.910,-104.660,5.090,0.0500,0.0800,1.0000
C00687=-66.080,-105.890,5.100,0.0400,0.0600,1.0000
C00688=-64.190,-107.110,5.100,0.0300,0.0400,1.0000
C00689=-61.780,-108.580,5.100,0.0100,0.0300,1.0000
C00690=-58.730,-110.300,5.100,0.0100,0.0100,1.0000
C00691=-55.410,-112.040,5.100,0.0000,0.0000,1.0000
C00692=-52.220,-113.570,5.100,0.0000,0.0000,1.0000
C00693=-49.280,-114.880,5.100,0.0000,0.0000,1.0000
C00694=-46.390,-116.070,5.100,0.0000,0.0000,1.0000
C00695=-43.380,-117.230,5.100,0.0000,0.0000,1.0000
C00696=-40.050,-118.400,5.100,0.0000,0.0000,1.0000
C00697=-36.470,-119.520,5.100,0.0000,0.0100,1.0000
C00698=-33.090,-120.460,5.100,0.0100,0.0300,1.0000
C00699=-30.350,-121.130,5.100,0.0100,0.0500,1.0000
C00700=-28.160,-121.600,5.100,0.0100,0.0700,1.0000
C00701=-25.990,-122.020,5.090,0.0200,0.0900,1.0000
C00702=-23.300,-122.520,5.090,0.0200,0.1100,0.9900
C00703=-19.390,-123.160,5.090,0.0200,0.1200,0.9900
C00704=-13.680,-123.910,5.090,0.0100,0.1300,0.9900
C00705=-7.210,-124.460,5.090,0.0100,0.1300,0.9900
C00706=0.000,-124.670,5.090,0.0000,0.1300,0.9900
C00707=0.000,-124.670,5.090,0.0000,0.1300,0.9900
C00708=7.210,-124.460,5.090,-0.0100,0.1300,0.9900
C00709=13.680,-123.910,5.090,-0.0100,0.1300,0.9900
C00710=19.390,-123.160,5.090,-0.0200,0.1200,0.9900
C00711=23.300,-122.520,5.090,-0.0200,0.1100,0.9900
C00712=25.990,-122.020,5.090,-0.0200,0.0900,1.0000
C00713=28.160,-121.600,5.100,-0.0100,0.0700,1.0000
C00714=30.350,-121.130,5.100,-0.0100,0.0500,1.0000
C00715=33.090,-120.460,5.100,-0.0100,0.0300,1.0000
C00716=36.470,-119.520,5.100,-0.0000,0.0100,1.0000
C00717=40.050,-118.400,5.100,-0.0000,0.0000,1.0000
C00718=43.380,-117.230,5.100,-0.0000,0.0000,1.0000
C00719=46.390,-116.070,5.100,-0.0000,0.0000,1.0000
C00720=49.280,-114.880,5.100,-0.0000,0.0000,1.0000
C00721=52.220,-113.570,5.100,-0.0000,0.0000,1.0000
C00722=55.410,-112.040,5.100,-0.0000,0.0000,1.0000
C00723=58.730,-110.300,5.100,-0.0100,0.0100,1.0000
C00724=61.780,-108.580,5.100,-0.0100,0.0300,1.0000
C00725=64.190,-107.110,5.100,-0.0300,0.0400,1.0000
C00726=66.080,-105.890,5.100,-0.0400,0.0600,1.0000
C00727=67.910,-104.660,5.090,-0.0500,0.0800,1.0000
C00728=70.160,-103.110,5.090,-0.0600,0.0900,0.9900
C00729=73.380,-100.800,5.090,-0.0700,0.1000,0.9900
C00730=77.940,-97.300,5.090,-0.0800,0.1000,0.9900
C00731=82.910,-93.100,5.090,-0.0900,0.1000,0.9900
C00732=88.150,-88.150,5.090,-0.0900,0.0900,0.9900
C00733=93.100,-82.910,5.090,-0.1000,0.0900,0.9900
C00734=97.300,-77.940,5.090,-0.1000,0.0800,0.9900
C00735=100.800,-73.380,5.090,-0.1000,0.0700,0.9900
C00736=103.110,-70.160,5.090,-0.0900,0.0600,0.9900
C00737=104.660,-67.910,5.090,-0.0800,0.0500,1.0000
C00738=105.890,-66.080,5.100,-0.0600,0.0400,1.0000
C00739=107.110,-64.190,5.100,-0.0400,0.0300,1.0000
C00740=108.580,-61.780,5.100,-0.0300,0.0100,1.0000
C00741=110.300,-58.730,5.100,-0.0100,0.0100,1.0000
C00742=112.040,-55.410,5.100,-0.0000,0.0000,1.0000
C00743=113.570,-52.220,5.100,-0.0000,0.0000,1.0000
C00744=114.880,-49.280,5.100,-0.0000,0.0000,1.0000
C00745=116.070,-46.390,5.100,-0.0000,0.0000,1.0000
C00746=117.230,-43.380,5.100,-0.0000,0.0000,1.0000
C00747=118.400,-40.050,5.100,-0.0000,0.0000,1.0000
C00748=119.520,-36.470,5.100,-0.0100,0.0000,1.0000
C00749=120.460,-33.090,5.100,-0.0300,0.0100,1.0000
C00750=121.130,-30.350,5.100,-0.0500,0.0100,1.0000
C00751=121.600,-28.160,5.100,-0.0700,0.0100,1.0000
C00752=122.020,-25.990,5.090,-0.0900,0.0200,1.0000
C00753=122.520,-23.300,5.090,-0.1100,0.0200,0.9900
C00754=123.160,-19.390,5.090,-0.1200,0.0200,0.9900
C00755=123.910,-13.680,5.090,-0.1300,0.0100,0.9900
C00756=124.460,-7.210,5.090,-0.1300,0.0100,0.9900
C00757=124.670,0.000,5.090,-0.1300,0.0000,0.9900
C00758=124.460,7.210,5.090,-0.1300,-0.0100,0.9900
C00759=123.910,13.680,5.090,-0.1300,-0.0100,0.9900
C00760=123.160,19.390,5.090,-0.1200,-0.0200,0.9900
C00761=122.520,23.300,5.090,-0.1100,-0.0200,0.9900
C00762=122.020,25.990,5.090,-0.0900,-0.0200,1.0000
C00763=121.600,28.160,5.100,-0.0700,-0.0100,1.0000
C00764=121.130,30.350,5.100,-0.0500,-0.0100,1.0000
C00765=120.460,33.090,5.100,-0.0300,-0.0100,1.0000
C00766=119.520,36.470,5.100,-0.0100,-0.0000,1.0000
C00767=118.400,40.050,5.100,-0.0000,-0.0000,1.0000
C00768=117.230,43.380,5.100,-0.0000,-0.0000,1.0000
C00769=116.070,46.390,5.100,-0.0000,-0.0000,1.0000
C00770=114.880,49.280,5.100,-0.0000,-0.0000,1.0000
C00771=113.570,52.220,5.100,-0.0000,-0.0000,1.0000
C00772=112.040,55.410,5.100,-0.0000,-0.0000,1.0000
C00773=110.300,58.730,5.100,-0.0100,-0.0100,1.0000
C00774=108.580,61.780,5.100,-0.0300,-0.0100,1.0000
C00775=107.110,64.190,5.100,-0.0400,-0.0300,1.0000
C00776=105.890,66.080,5.100,-0.0600,-0.0400,1.0000
C00777=104.660,67.910,5.090,-0.0800,-0.0500,1.0000
C00778=103.110,70.160,5.090,-0.0900,-0.0600,0.9900
C00779=100.800,73.380,5.090,-0.1000,-0.0700,0.9900
C00780=97.300,77.940,5.090,-0.1000,-0.0800,0.9900
C00781=93.100,82.910,5.090,-0.1000,-0.0900,0.9900
C00782=88.150,88.150,5.090,-0.0900,-0.0900,0.9900
C00783=82.910,93.100,5.090,-0.0900,-0.1000,0.9900
C00784=77.940,97.300,5.090,-0.0800,-0.1000,0.9900
C00785=73.380,100.800,5.090,-0.0700,-0.1000,0.9900
C00786=70.160,103.110,5.090,-0.0600,-0.0900,0.9900
C00787=67.910,104.660,5.090,-0.0500,-0.0800,1.0000
C00788=66.080,105.890,5.100,-0.0400,-0.0600,1.0000
C00789=64.190,107.110,5.100,-0.0300,-0.0400,1.0000
C00790=61.780,108.580,5.100,-0.0100,-0.0300,1.0000
C00791=58.730,110.300,5.100,-0.0100,-0.0100,1.0000
C00792=55.410,112.040,5.100,-0.0000,-0.0000,1.0000
C00793=52.220,113.570,5.100,-0.0000,-0.0000,1.0000
C00794=49.280,114.880,5.100,-0.0000,-0.0000,1.0000
C00795=46.390,116.070,5.100,-0.0000,-0.0000,1.0000
C00796=43.380,117.230,5.100,-0.0000,-0.0000,1.0000
C00797=40.050,118.400,5.100,-0.0000,-0.0000,1.0000
C00798=36.470,119.520,5.100,-0.0000,-0.0100,1.0000
C00799=33.090,120.460,5.100,-0.0100,-0.0300,1.0000
C00800=30.350,121.130,5.100,-0.0100,-0.0500,1.0000
C00801=28.160,121.600,5.100,-0.0100,-0.0700,1.0000
C00802=25.990,122.020,5.090,-0.0200,-0.0900,1.0000
C00803=23.300,122.520,5.090,-0.0200,-0.1100,0.9900
C00804=19.390,123.160,5.090,-0.0200,-0.1200,0.9900
C00805=13.680,123.910,5.090,-0.0100,-0.1300,0.9900
C00806=7.210,124.460,5.090,-0.0100,-0.1300,0.9900
C00807=0.000,124.670,5.090,0.0000,-0.1300,0.9900
C00808=0.000,124.420,6.770,0.0000,-0.1700,0.9900
C00809=7.190,124.210,6.770,-0.0100,-0.1700,0.9900
C00810=13.650,123.670,6.770,-0.0200,-0.1700,0.9900
C00811=19.350,122.930,6.770,-0.0200,-0.1600,0.9900
C00812=23.240,122.310,6.780,-0.0200,-0.1400,0.9900
C00813=25.920,121.850,6.780,-0.0200,-0.1200,0.9900
C00814=28.090,121.470,6.790,-0.0200,-0.0900,1.0000
C00815=30.280,121.050,6.790,-0.0100,-0.0600,1.0000
C00816=33.020,120.420,6.800,-0.0100,-0.0400,1.0000
C00817=36.400,119.510,6.800,-0.0000,-0.0200,1.0000
C00818=39.990,118.410,6.800,-0.0000,-0.0000,1.0000
C00819=43.340,117.240,6.800,-0.0000,-0.0000,1.0000
C00820=46.370,116.080,6.800,-0.0000,-0.0000,1.0000
C00821=49.290,114.870,6.800,-0.0000,-0.0000,1.0000
C00822=52.250,113.550,6.800,-0.0000,-0.0000,1.0000
C00823=55.450,112.010,6.800,-0.0000,-0.0000,1.0000
C00824=58.770,110.250,6.800,-0.0100,-0.0200,1.0000
C00825=61.800,108.500,6.800,-0.0200,-0.0300,1.0000
C00826=64.180,107.010,6.790,-0.0300,-0.0500,1.0000
C00827=66.030,105.760,6.790,-0.0500,-0.0700,1.0000
C00828=67.830,104.490,6.780,-0.0700,-0.1000,0.9900
C00829=70.050,102.920,6.780,-0.0800,-0.1200,0.9900
C00830=73.240,100.600,6.770,-0.1000,-0.1300,0.9900
C00831=77.800,97.090,6.770,-0.1000,-0.1300,0.9900
C00832=82.750,92.910,6.770,-0.1100,-0.1200,0.9900
C00833=87.980,87.980,6.770,-0.1200,-0.1200,0.9900
C00834=92.910,82.750,6.770,-0.1200,-0.1100,0.9900
C00835=97.090,77.800,6.770,-0.1300,-0.1000,0.9900
C00836=100.600,73.240,6.770,-0.1300,-0.1000,0.9900
C00837=102.920,70.050,6.780,-0.1200,-0.0800,0.9900
C00838=104.490,67.830,6.780,-0.1000,-0.0700,0.9900
C00839=105.760,66.030,6.790,-0.0700,-0.0500,1.0000
C00840=107.010,64.180,6.790,-0.0500,-0.0300,1.0000
C00841=108.500,61.800,6.800,-0.0300,-0.0200,1.0000
C00842=110.250,58.770,6.800,-0.0200,-0.0100,1.0000
C00843=112.010,55.450,6.800,-0.0000,-0.0000,1.0000
C00844=113.550,52.250,6.800,-0.0000,-0.0000,1.0000
C00845=114.870,49.290,6.800,-0.0000,-0.0000,1.0000
C00846=116.080,46.370,6.800,-0.0000,-0.0000,1.0000
C00847=117.240,43.340,6.800,-0.0000,-0.0000,1.0000
C00848=118.410,39.990,6.800,-0.0000,-0.0000,1.0000
C00849=119.510,36.400,6.800,-0.0200,-0.0000,1.0000
C00850=120.420,33.020,6.800,-0.0400,-0.0100,1.0000
C00851=121.050,30.280,6.790,-0.0600,-0.0100,1.0000
C00852=121.470,28.090,6.790,-0.0900,-0.0200,1.0000
C00853=121.850,25.920,6.780,-0.1200,-0.0200,0.9900
C00854=122.310,23.240,6.780,-0.1400,-0.0200,0.9900
C00855=122.930,19.350,6.770,-0.1600,-0.0200,0.9900
C00856=123.670,13.650,6.770,-0.1700,-0.0200,0.9900
C00857=124.210,7.190,6.770,-0.1700,-0.0100,0.9900
C00858=124.420,0.000,6.770,-0.1700,0.0000,0.9900
C00859=124.210,-7.190,6.770,-0.1700,0.0100,0.9900
C00860=123.670,-13.650,6.770,-0.1700,0.0200,0.9900
C00861=122.930,-19.350,6.770,-0.1600,0.0200,0.9900
C00862=122.310,-23.240,6.780,-0.1400,0.0200,0.9900
C00863=121.850,-25.920,6.780,-0.1200,0.0200,0.9900
C00864=121.470,-28.090,6.790,-0.0900,0.0200,1.0000
C00865=121.050,-30.280,6.790,-0.0600,0.0100,1.0000
C00866=120.420,-33.020,6.800,-0.0400,0.0100,1.0000
C00867=119.510,-36.400,6.800,-0.0200,0.0000,1.0000
C00868=118.410,-39.990,6.800,-0.0000,0.0000,1.0000
C00869=117.240,-43.340,6.800,-0.0000,0.0000,1.0000
C00870=116.080,-46.370,6.800,-0.0000,0.0000,1.0000
C00871=114.870,-49.290,6.800,-0.0000,0.0000,1.0000
C00872=113.550,-52.250,6.800,-0.0000,0.0000,1.0000
C00873=112.010,-55.450,6.800,-0.0000,0.0000,1.0000
C00874=110.250,-58.770,6.800,-0.0200,0.0100,1.0000
C00875=108.500,-61.800,6.800,-0.0300,0.0200,1.0000
C00876=107.010,-64.180,6.790,-0.0500,0.0300,1.0000
C00877=105.760,-66.030,6.790,-0.0700,0.0500,1.0000
C00878=104.490,-67.830,6.780,-0.1000,0.0700,0.9900
C00879=102.920,-70.050,6.780,-0.1200,0.0800,0.9900
C00880=100.600,-73.240,6.770,-0.1300,0.1000,0.9900
C00881=97.090,-77.800,6.770,-0.1300,0.1000,0.9900
C00882=92.910,-82.750,6.770,-0.1200,0.1100,0.9900
C00883=87.980,-87.980,6.770,-0.1200,0.1200,0.9900
C00884=82.750,-92.910,6.770,-0.1100,0.1200,0.9900
C00885=77.800,-97.090,6.770,-0.1000,0.1300,0.9900
C00886=73.240,-100.600,6.770,-0.1000,0.1300,0.9900
C00887=70.050,-102.920,6.780,-0.0800,0.1200,0.9900
C00888=67.830,-104.490,6.780,-0.0700,0.1000,0.9900
C00889=66.030,-105.760,6.790,-0.0500,0.0700,1.0000
C00890=64.180,-107.010,6.790,-0.0300,0.0500,1.0000
C00891=61.800,-108.500,6.800,-0.0200,0.0300,1.0000
C00892=58.770,-110.250,6.800,-0.0100,0.0200,1.0000
C00893=55.450,-112.010,6.800,-0.0000,0.0000,1.0000
C00894=52.250,-113.550,6.800,-0.0000,0.0000,1.0000
C00895=49.290,-114.870,6.800,-0.0000,0.0000,1.0000
C00896=46.370,-116.080,6.800,-0.0000,0.0000,1.0000
C00897=43.340,-117.240,6.800,-0.0000,0.0000,1.0000
C00898=39.990,-118.410,6.800,-0.0000,0.0000,1.0000
C00899=36.400,-119.510,6.800,-0.0000,0.0200,1.0000
C00900=33.020,-120.420,6.800,-0.0100,0.0400,1.0000
C00901=30.280,-121.050,6.790,-0.0100,0.0600,1.0000
C00902=28.090,-121.470,6.790,-0.0200,0.0900,1.0000
C00903=25.920,-121.850,6.780,-0.0200,0.1200,0.9900
C00904=23.240,-122.310,6.780,-0.0200,0.1400,0.9900
C00905=19.350,-122.930,6.770,-0.0200,0.1600,0.9900
C00906=13.650,-123.670,6.770,-0.0200,0.1700,0.9900
C00907=7.190,-124.210,6.770,-0.0100,0.1700,0.9900
C00908=0.000,-124.420,6.770,0.0000,0.1700,0.9900
C00909=0.000,-124.420,6.770,0.0000,0.1700,0.9900
C00910=-7.190,-124.210,6.770,0.0100,0.1700,0.9900
C00911=-13.650,-123.670,6.770,0.0200,0.1700,0.9900
C00912=-19.350,-122.930,6.770,0.0200,0.1600,0.9900
C00913=-23.240,-122.310,6.780,0.0200,0.1400,0.9900
C00914=-25.920,-121.850,6.780,0.0200,0.1200,0.9900
C00915=-28.090,-121.470,6.790,0.0200,0.0900,1.0000
C00916=-30.280,-121.050,6.790,0.0100,0.0600,1.0000
C00917=-33.020,-120.420,6.800,0.0100,0.0400,1.0000
C00918=-36.400,-119.510,6.800,0.0000,0.0200,1.0000
C00919=-39.990,-118.410,6.800,0.0000,0.0000,1.0000
C00920=-43.340,-117.240,6.800,0.0000,0.0000,1.0000
C00921=-46.370,-116.080,6.800,0.0000,0.0000,1.0000
C00922=-49.290,-114.870,6.800,0.0000,0.0000,1.0000
C00923=-52.250,-113.550,6.800,0.0000,0.0000,1.0000
C00924=-55.450,-112.010,6.800,0.0000,0.0000,1.0000
C00925=-58.770,-110.250,6.800,0.0100,0.0200,1.0000
C00926=-61.800,-108.500,6.800,0.0200,0.0300,1.0000
C00927=-64.180,-107.010,6.790,0.0300,0.0500,1.0000
C00928=-66.030,-105.760,6.790,0.0500,0.0700,1.0000
C00929=-67.830,-104.490,6.780,0.0700,0.1000,0.9900
C00930=-70.050,-102.920,6.780,0.0800,0.1200,0.9900
C00931=-73.240,-100.600,6.770,0.1000,0.1300,0.9900
C00932=-77.800,-97.090,6.770,0.1000,0.1300,0.9900
C00933=-82.750,-92.910,6.770,0.1100,0.1200,0.9900
C00934=-87.980,-87.980,6.770,0.1200,0.1200,0.9900
C00935=-92.910,-82.750,6.770,0.1200,0.1100,0.9900
C00936=-97.090,-77.800,6.770,0.1300,0.1000,0.9900
C00937=-100.600,-73.240,6.770,0.1300,0.1000,0.9900
C00938=-102.920,-70.050,6.780,0.1200,0.0800,0.9900
C00939=-104.490,-67.830,6.780,0.1000,0.0700,0.9900
C00940=-105.760,-66.030,6.790,0.0700,0.0500,1.0000
C00941=-107.010,-64.180,6.790,0.0500,0.0300,1.0000
C00942=-108.500,-61.800,6.800,0.0300,0.0200,1.0000
C00943=-110.250,-58.770,6.800,0.0200,0.0100,1.0000
C00944=-112.010,-55.450,6.800,0.0000,0.0000,1.0000
C00945=-113.550,-52.250,6.800,0.0000,0.0000,1.0000
C00946=-114.870,-49.290,6.800,0.0000,0.0000,1.0000
C00947=-116.080,-46.370,6.800,0.0000,0.0000,1.0000
C00948=-117.240,-43.340,6.800,0.0000,0.0000,1.0000
C00949=-118.410,-39.990,6.800,0.0000,0.0000,1.0000
C00950=-119.510,-36.400,6.800,0.0200,0.0000,1.0000
C00951=-120.420,-33.020,6.800,0.0400,0.0100,1.0000
C00952=-121.050,-30.280,6.790,0.0600,0.0100,1.0000
C00953=-121.470,-28.090,6.790,0.0900,0.0200,1.0000
C00954=-121.850,-25.920,6.780,0.1200,0.0200,0.9900
C00955=-122.310,-23.240,6.780,0.1400,0.0200,0.9900
C00956=-122.930,-19.350,6.770,0.1600,0.0200,0.9900
C00957=-123.670,-13.650,6.770,0.1700,0.0200,0.9900
C00958=-124.210,-7.190,6.770,0.1700,0.0100,0.9900
C00959=-124.420,0.000,6.770,0.1700,-0.0000,0.9900
C00960=-124.210,7.190,6.770,0.1700,-0.0100,0.9900
C00961=-123.670,13.650,6.770,0.1700,-0.0200,0.9900
C00962=-122.930,19.350,6.770,0.1600,-0.0200,0.9900
C00963=-122.310,23.240,6.780,0.1400,-0.0200,0.9900
C00964=-121.850,25.920,6.780,0.1200,-0.0200,0.9900
C00965=-121.470,28.090,6.790,0.0900,-0.0200,1.0000
C00966=-121.050,30.280,6.790,0.0600,-0.0100,1.0000
C00967=-120.420,33.020,6.800,0.0400,-0.0100,1.0000
C00968=-119.510,36.400,6.800,0.0200,-0.0000,1.0000
C00969=-118.410,39.990,6.800,0.0000,-0.0000,1.0000
C00970=-117.240,43.340,6.800,0.0000,-0.0000,1.0000
C00971=-116.080,46.370,6.800,0.0000,-0.0000,1.0000
C00972=-114.870,49.290,6.800,0.0000,-0.0000,1.0000
C00973=-113.550,52.250,6.800,0.0000,-0.0000,1.0000
C00974=-112.010,55.450,6.800,0.0000,-0.0000,1.0000
C00975=-110.250,58.770,6.800,0.0200,-0.0100,1.0000
C00976=-108.500,61.800,6.800,0.0300,-0.0200,1.0000
C00977=-107.010,64.180,6.790,0.0500,-0.0300,1.0000
C00978=-105.760,66.030,6.790,0.0700,-0.0500,1.0000
C00979=-104.490,67.830,6.780,0.1000,-0.0700,0.9900
C00980=-102.920,70.050,6.780,0.1200,-0.0800,0.9900
C00981=-100.600,73.240,6.770,0.1300,-0.1000,0.9900
C00982=-97.090,77.800,6.770,0.1300,-0.1000,0.9900
C00983=-92.910,82.750,6.770,0.1200,-0.1100,0.9900
C00984=-87.980,87.980,6.770,0.1200,-0.1200,0.9900
C00985=-82.750,92.910,6.770,0.1100,-0.1200,0.9900
C00986=-77.800,97.090,6.770,0.1000,-0.1300,0.9900
C00987=-73.240,100.600,6.770,0.1000,-0.1300,0.9900
C00988=-70.050,102.920,6.780,0.0800,-0.1200,0.9900
C00989=-67.830,104.490,6.780,0.0700,-0.1000,0.9900
C00990=-66.030,105.760,6.790,0.0500,-0.0700,1.0000
C00991=-64.180,107.010,6.790,0.0300,-0.0500,1.0000
C00992=-61.800,108.500,6.800,0.0200,-0.0300,1.0000
C00993=-58.770,110.250,6.800,0.0100,-0.0200,1.0000
C00994=-55.450,112.010,6.800,0.0000,-0.0000,1.0000
C00995=-52.250,113.550,6.800,0.0000,-0.0000,1.0000
C00996=-49.290,114.870,6.800,0.0000,-0.0000,1.0000
C00997=-46.370,116.080,6.800,0.0000,-0.0000,1.0000
C00998=-43.340,117.240,6.800,0.0000,-0.0000,1.0000
C00999=-39.990,118.410,6.800,0.0000,-0.0000,1.0000
C01000=-36.400,119.510,6.800,0.0000,-0.0200,1.0000
C01001=-33.020,120.420,6.800,0.0100,-0.0400,1.0000
C01002=-30.280,121.050,6.790,0.0100,-0.0600,1.0000
C01003=-28.090,121.470,6.790,0.0200,-0.0900,1.0000
C01004=-25.920,121.850,6.780,0.0200,-0.1200,0.9900
C01005=-23.240,122.310,6.780,0.0200,-0.1400,0.9900
C01006=-19.350,122.930,6.770,0.0200,-0.1600,0.9900
C01007=-13.650,123.670,6.770,0.0200,-0.1700,0.9900
C01008=-7.190,124.210,6.770,0.0100,-0.1700,0.9900
C01009=0.000,124.420,6.770,0.0000,-0.1700,0.9900
C01010=0.000,124.100,8.440,0.0000,-0.2000,0.9800
C01011=-7.160,123.890,8.440,0.0100,-0.2000,0.9800
C01012=-13.600,123.350,8.440,0.0200,-0.2000,0.9800
C01013=-19.290,122.630,8.440,0.0300,-0.1900,0.9800
C01014=-23.170,122.040,8.450,0.0300,-0.1700,0.9800
C01015=-25.850,121.640,8.470,0.0200,-0.1400,0.9900
C01016=-28.010,121.310,8.480,0.0200,-0.1100,0.9900
C01017=-30.190,120.950,8.490,0.0100,-0.0700,1.0000
C01018=-32.920,120.370,8.490,0.0100,-0.0400,1.0000
C01019=-36.310,119.500,8.500,0.0100,-0.0200,1.0000
C01020=-39.920,118.420,8.500,0.0000,-0.0100,1.0000
C01021=-43.300,117.260,8.500,0.0000,-0.0000,1.0000
C01022=-46.360,116.080,8.500,0.0000,-0.0000,1.0000
C01023=-49.300,114.870,8.500,0.0000,-0.0000,1.0000
C01024=-52.290,113.530,8.500,0.0000,-0.0000,1.0000
C01025=-55.510,111.970,8.500,0.0000,-0.0100,1.0000
C01026=-58.830,110.180,8.500,0.0100,-0.0200,1.0000
C01027=-61.830,108.400,8.490,0.0200,-0.0400,1.0000
C01028=-64.170,106.870,8.490,0.0400,-0.0600,1.0000
C01029=-65.980,105.590,8.480,0.0700,-0.0900,0.9900
C01030=-67.730,104.290,8.470,0.0900,-0.1200,0.9900
C01031=-69.910,102.680,8.450,0.1000,-0.1400,0.9800
C01032=-73.070,100.350,8.440,0.1200,-0.1600,0.9800
C01033=-77.610,96.840,8.440,0.1300,-0.1600,0.9800
C01034=-82.540,92.670,8.440,0.1400,-0.1500,0.9800
C01035=-87.750,87.750,8.440,0.1400,-0.1400,0.9800
C01036=-92.670,82.540,8.440,0.1500,-0.1400,0.9800
C01037=-96.840,77.610,8.440,0.1600,-0.1300,0.9800
C01038=-100.350,73.070,8.440,0.1600,-0.1200,0.9800
C01039=-102.680,69.910,8.450,0.1400,-0.1000,0.9800
C01040=-104.290,67.730,8.470,0.1200,-0.0900,0.9900
C01041=-105.590,65.980,8.480,0.0900,-0.0700,0.9900
C01042=-106.870,64.170,8.490,0.0600,-0.0400,1.0000
C01043=-108.400,61.830,8.490,0.0400,-0.0200,1.0000
C01044=-110.180,58.830,8.500,0.0200,-0.0100,1.0000
C01045=-111.970,55.510,8.500,0.0100,-0.0000,1.0000
C01046=-113.530,52.290,8.500,0.0000,-0.0000,1.0000
C01047=-114.870,49.300,8.500,0.0000,-0.0000,1.0000
C01048=-116.080,46.360,8.500,0.0000,-0.0000,1.0000
C01049=-117.260,43.300,8.500,0.0000,-0.0000,1.0000
C01050=-118.420,39.920,8.500,0.0100,-0.0000,1.0000
C01051=-119.500,36.310,8.500,0.0200,-0.0100,1.0000
C01052=-120.370,32.920,8.490,0.0400,-0.0100,1.0000
C01053=-120.950,30.190,8.490,0.0700,-0.0100,1.0000
C01054=-121.310,28.010,8.480,0.1100,-0.0200,0.9900
C01055=-121.640,25.850,8.470,0.1400,-0.0200,0.9900
C01056=-122.040,23.170,8.450,0.1700,-0.0300,0.9800
C01057=-122.630,19.290,8.440,0.1900,-0.0300,0.9800
C01058=-123.350,13.600,8.440,0.2000,-0.0200,0.9800
C01059=-123.890,7.160,8.440,0.2000,-0.0100,0.9800
C01060=-124.100,0.000,8.440,0.2000,-0.0000,0.9800
C01061=-123.890,-7.160,8.440,0.2000,0.0100,0.9800
C01062=-123.350,-13.600,8.440,0.2000,0.0200,0.9800
C01063=-122.630,-19.290,8.440,0.1900,0.0300,0.9800
C01064=-122.040,-23.170,8.450,0.1700,0.0300,0.9800
C01065=-121.640,-25.850,8.470,0.1400,0.0200,0.9900
C01066=-121.310,-28.010,8.480,0.1100,0.0200,0.9900
C01067=-120.950,-30.190,8.490,0.0700,0.0100,1.0000
C01068=-120.370,-32.920,8.490,0.0400,0.0100,1.0000
C01069=-119.500,-36.310,8.500,0.0200,0.0100,1.0000
C01070=-118.420,-39.920,8.500,0.0100,0.0000,1.0000
C01071=-117.260,-43.300,8.500,0.0000,0.0000,1.0000
C01072=-116.080,-46.360,8.500,0.0000,0.0000,1.0000
C01073=-114.870,-49.300,8.500,0.0000,0.0000,1.0000
C01074=-113.530,-52.290,8.500,0.0000,0.0000,1.0000
C01075=-111.970,-55.510,8.500,0.0100,0.0000,1.0000
C01076=-110.180,-58.830,8.500,0.0200,0.0100,1.0000
C01077=-108.400,-61.830,8.490,0.0400,0.0200,1.0000
C01078=-106.870,-64.170,8.490,0.0600,0.0400,1.0000
C01079=-105.590,-65.980,8.480,0.0900,0.0700,0.9900
C01080=-104.290,-67.730,8.470,0.1200,0.0900,0.9900
C01081=-102.680,-69.910,8.450,0.1400,0.1000,0.9800
C01082=-100.350,-73.070,8.440,0.1600,0.1200,0.9800
C01083=-96.840,-77.610,8.440,0.1600,0.1300,0.9800
C01084=-92.670,-82.540,8.440,0.1500,0.1400,0.9800
C01085=-87.750,-87.750,8.440,0.1400,0.1400,0.9800
C01086=-82.540,-92.670,8.440,0.1400,0.1500,0.9800
C01087=-77.610,-96.840,8.440,0.1300,0.1600,0.9800
C01088=-73.070,-100.350,8.440,0.1200,0.1600,0.9800
C01089=-69.910,-102.680,8.450,0.1000,0.1400,0.9800
C01090=-67.730,-104.290,8.470,0.0900,0.1200,0.9900
C01091=-65.980,-105.590,8.480,0.0700,0.0900,0.9900
C01092=-64.170,-106.870,8.490,0.0400,0.0600,1.0000
C01093=-61.830,-108.400,8.490,0.0200,0.0400,1.0000
C01094=-58.830,-110.180,8.500,0.0100,0.0200,1.0000
C01095=-55.510,-111.970,8.500,0.0000,0.0100,1.0000
C01096=-52.290,-113.530,8.500,0.0000,0.0000,1.0000
C01097=-49.300,-114.870,8.500,0.0000,0.0000,1.0000
C01098=-46.360,-116.080,8.500,0.0000,0.0000,1.0000
C01099=-43.300,-117.260,8.500,0.0000,0.0000,1.0000
C01100=-39.920,-118.420,8.500,0.0000,0.0100,1.0000
C01101=-36.310,-119.500,8.500,0.0100,0.0200,1.0000
C01102=-32.920,-120.370,8.490,0.0100,0.0400,1.0000
C01103=-30.190,-120.950,8.490,0.0100,0.0700,1.0000
C01104=-28.010,-121.310,8.480,0.0200,0.1100,0.9900
C01105=-25.850,-121.640,8.470,0.0200,0.1400,0.9900
C01106=-23.170,-122.040,8.450,0.0300,0.1700,0.9800
C01107=-19.290,-122.630,8.440,0.0300,0.1900,0.9800
C01108=-13.600,-123.350,8.440,0.0200,0.2000,0.9800
C01109=-7.160,-123.890,8.440,0.0100,0.2000,0.9800
C01110=0.000,-124.100,8.440,0.0000,0.2000,0.9800
C01111=0.000,-124.100,8.440,0.0000,0.2000,0.9800
C01112=7.160,-123.890,8.440,-0.0100,0.2000,0.9800
C01113=13.600,-123.350,8.440,-0.0200,0.2000,0.9800
C01114=19.290,-122.630,8.440,-0.0300,0.1900,0.9800
C01115=23.170,-122.040,8.450,-0.0300,0.1700,0.9800
C01116=25.850,-121.640,8.470,-0.0200,0.1400,0.9900
C01117=28.010,-121.310,8.480,-0.0200,0.1100,0.9900
C01118=30.190,-120.950,8.490,-0.0100,0.0700,1.0000
C01119=32.920,-120.370,8.490,-0.0100,0.0400,1.0000
C01120=36.310,-119.500,8.500,-0.0100,0.0200,1.0000
C01121=39.920,-118.420,8.500,-0.0000,0.0100,1.0000
C01122=43.300,-117.260,8.500,-0.0000,0.0000,1.0000
C01123=46.360,-116.080,8.500,-0.0000,0.0000,1.0000
C01124=49.300,-114.870,8.500,-0.0000,0.0000,1.0000
C01125=52.290,-113.530,8.500,-0.0000,0.0000,1.0000
C01126=55.510,-111.970,8.500,-0.0000,0.0100,1.0000
C01127=58.830,-110.180,8.500,-0.0100,0.0200,1.0000
C01128=61.830,-108.400,8.490,-0.0200,0.0400,1.0000
C01129=64.170,-106.870,8.490,-0.0400,0.0600,1.0000
C01130=65.980,-105.590,8.480,-0.0700,0.0900,0.9900
C01131=67.730,-104.290,8.470,-0.0900,0.1200,0.9900
C01132=69.910,-102.680,8.450,-0.1000,0.1400,0.9800
C01133=73.070,-100.350,8.440,-0.1200,0.1600,0.9800
C01134=77.610,-96.840,8.440,-0.1300,0.1600,0.9800
C01135=82.540,-92.670,8.440,-0.1400,0.1500,0.9800
C01136=87.750,-87.750,8.440,-0.1400,0.1400,0.9800
C01137=92.670,-82.540,8.440,-0.1500,0.1400,0.9800
C01138=96.840,-77.610,8.440,-0.1600,0.1300,0.9800
C01139=100.350,-73.070,8.440,-0.1600,0.1200,0.9800
C01140=102.680,-69.910,8.450,-0.1400,0.1000,0.9800
C01141=104.290,-67.730,8.470,-0.1200,0.0900,0.9900
C01142=105.590,-65.980,8.480,-0.0900,0.0700,0.9900
C01143=106.870,-64.170,8.490,-0.0600,0.0400,1.0000
C01144=108.400,-61.830,8.490,-0.0400,0.0200,1.0000
C01145=110.180,-58.830,8.500,-0.0200,0.0100,1.0000
C01146=111.970,-55.510,8.500,-0.0100,0.0000,1.0000
C01147=113.530,-52.290,8.500,-0.0000,0.0000,1.0000
C01148=114.870,-49.300,8.500,-0.0000,0.0000,1.0000
C01149=116.080,-46.360,8.500,-0.0000,0.0000,1.0000
C01150=117.260,-43.300,8.500,-0.0000,0.0000,1.0000
C01151=118.420,-39.920,8.500,-0.0100,0.0000,1.0000
C01152=119.500,-36.310,8.500,-0.0200,0.0100,1.0000
C01153=120.370,-32.920,8.490,-0.0400,0.0100,1.0000
C01154=120.950,-30.190,8.490,-0.0700,0.0100,1.0000
C01155=121.310,-28.010,8.480,-0.1100,0.0200,0.9900
C01156=121.640,-25.850,8.470,-0.1400,0.0200,0.9900
C01157=122.040,-23.170,8.450,-0.1700,0.0300,0.9800
C01158=122.630,-19.290,8.440,-0.1900,0.0300,0.9800
C01159=123.350,-13.600,8.440,-0.2000,0.0200,0.9800
C01160=123.890,-7.160,8.440,-0.2000,0.0100,0.9800
C01161=124.100,0.000,8.440,-0.2000,0.0000,0.9800
C01162=123.890,7.160,8.440,-0.2000,-0.0100,0.9800
C01163=123.350,13.600,8.440,-0.2000,-0.0200,0.9800
C01164=122.630,19.290,8.440,-0.1900,-0.0300,0.9800
C01165=122.040,23.170,8.450,-0.1700,-0.0300,0.9800
C01166=121.640,25.850,8.470,-0.1400,-0.0200,0.9900
C01167=121.310,28.010,8.480,-0.1100,-0.0200,0.9900
C01168=120.950,30.190,8.490,-0.0700,-0.0100,1.0000
C01169=120.370,32.920,8.490,-0.0400,-0.0100,1.0000
C01170=119.500,36.310,8.500,-0.0200,-0.0100,1.0000
C01171=118.420,39.920,8.500,-0.0100,-0.0000,1.0000
C01172=117.260,43.300,8.500,-0.0000,-0.0000,1.0000
C01173=116.080,46.360,8.500,-0.0000,-0.0000,1.0000
C01174=114.870,49.300,8.500,-0.0000,-0.0000,1.0000
C01175=113.530,52.290,8.500,-0.0000,-0.0000,1.0000
C01176=111.970,55.510,8.500,-0.0100,-0.0000,1.0000
C01177=110.180,58.830,8.500,-0.0200,-0.0100,1.0000
C01178=108.400,61.830,8.490,-0.0400,-0.0200,1.0000
C01179=106.870,64.170,8.490,-0.0600,-0.0400,1.0000
C01180=105.590,65.980,8.480,-0.0900,-0.0700,0.9900
C01181=104.290,67.730,8.470,-0.1200,-0.0900,0.9900
C01182=102.680,69.910,8.450,-0.1400,-0.1000,0.9800
C01183=100.350,73.070,8.440,-0.1600,-0.1200,0.9800
C01184=96.840,77.610,8.440,-0.1600,-0.1300,0.9800
C01185=92.670,82.540,8.440,-0.1500,-0.1400,0.9800
C01186=87.750,87.750,8.440,-0.1400,-0.1400,0.9800
C01187=82.540,92.670,8.440,-0.1400,-0.1500,0.9800
C01188=77.610,96.840,8.440,-0.1300,-0.1600,0.9800
C01189=73.070,100.350,8.440,-0.1200,-0.1600,0.9800
C01190=69.910,102.680,8.450,-0.1000,-0.1400,0.9800
C01191=67.730,104.290,8.470,-0.0900,-0.1200,0.9900
C01192=65.980,105.590,8.480,-0.0700,-0.0900,0.9900
C01193=64.170,106.870,8.490,-0.0400,-0.0600,1.0000
C01194=61.830,108.400,8.490,-0.0200,-0.0400,1.0000
C01195=58.830,110.180,8.500,-0.0100,-0.0200,1.0000
C01196=55.510,111.970,8.500,-0.0000,-0.0100,1.0000
C01197=52.290,113.530,8.500,-0.0000,-0.0000,1.0000
C01198=49.300,114.870,8.500,-0.0000,-0.0000,1.0000
C01199=46.360,116.080,8.500,-0.0000,-0.0000,1.0000
C01200=43.300,117.260,8.500,-0.0000,-0.0000,1.0000
C01201=39.920,118.420,8.500,-0.0000,-0.0100,1.0000
C01202=36.310,119.500,8.500,-0.0100,-0.0200,1.0000
C01203=32.920,120.370,8.490,-0.0100,-0.0400,1.0000
C01204=30.190,120.950,8.490,-0.0100,-0.0700,1.0000
C01205=28.010,121.310,8.480,-0.0200,-0.1100,0.9900
C01206=25.850,121.640,8.470,-0.0200,-0.1400,0.9900
C01207=23.170,122.040,8.450,-0.0300,-0.1700,0.9800
C01208=19.290,122.630,8.440,-0.0300,-0.1900,0.9800
C01209=13.600,123.350,8.440,-0.0200,-0.2000,0.9800
C01210=7.160,123.890,8.440,-0.0100,-0.2000,0.9800
C01211=0.000,124.100,8.440,0.0000,-0.2000,0.9800
C01212=0.000,123.720,10.100,0.0000,-0.2400,0.9700
C01213=7.120,123.520,10.100,-0.0100,-0.2400,0.9700
C01214=13.540,122.980,10.100,-0.0300,-0.2400,0.9700
C01215=19.220,122.270,10.100,-0.0300,-0.2300,0.9700
C01216=23.090,121.730,10.120,-0.0300,-0.2000,0.9800
C01217=25.750,121.380,10.140,-0.0200,-0.1700,0.9900
C01218=27.910,121.120,10.170,-0.0200,-0.1300,0.9900
C01219=30.090,120.820,10.180,-0.0100,-0.0900,1.0000
C01220=32.810,120.310,10.190,-0.0100,-0.0500,1.0000
C01221=36.210,119.490,10.190,-0.0100,-0.0200,1.0000
C01222=39.840,118.440,10.190,-0.0000,-0.0100,1.0000
C01223=43.250,117.270,10.200,-0.0000,-0.0000,1.0000
C01224=46.340,116.090,10.200,-0.0000,-0.0000,1.0000
C01225=49.320,114.860,10.200,-0.0000,-0.0000,1.0000
C01226=52.340,113.510,10.200,-0.0000,-0.0000,1.0000
C01227=55.580,111.920,10.190,-0.0000,-0.0100,1.0000
C01228=58.890,110.100,10.190,-0.0100,-0.0200,1.0000
C01229=61.870,108.270,10.190,-0.0300,-0.0400,1.0000
C01230=64.160,106.710,10.180,-0.0500,-0.0700,1.0000
C01231=65.910,105.380,10.170,-0.0800,-0.1000,0.9900
C01232=67.620,104.040,10.140,-0.1100,-0.1300,0.9900
C01233=69.750,102.400,10.120,-0.1200,-0.1600,0.9800
C01234=72.870,100.050,10.100,-0.1400,-0.1800,0.9700
C01235=77.390,96.540,10.100,-0.1500,-0.1900,0.9700
C01236=82.300,92.380,10.100,-0.1600,-0.1800,0.9700
C01237=87.490,87.490,10.100,-0.1700,-0.1700,0.9700
C01238=92.380,82.300,10.100,-0.1800,-0.1600,0.9700
C01239=96.540,77.390,10.100,-0.1900,-0.1500,0.9700
C01240=100.050,72.870,10.100,-0.1800,-0.1400,0.9700
C01241=102.400,69.750,10.120,-0.1600,-0.1200,0.9800
C01242=104.040,67.620,10.140,-0.1300,-0.1100,0.9900
C01243=105.380,65.910,10.170,-0.1000,-0.0800,0.9900
C01244=106.710,64.160,10.180,-0.0700,-0.0500,1.0000
C01245=108.270,61.870,10.190,-0.0400,-0.0300,1.0000
C01246=110.100,58.890,10.190,-0.0200,-0.0100,1.0000
C01247=111.920,55.580,10.190,-0.0100,-0.0000,1.0000
C01248=113.510,52.340,10.200,-0.0000,-0.0000,1.0000
C01249=114.860,49.320,10.200,-0.0000,-0.0000,1.0000
C01250=116.090,46.340,10.200,-0.0000,-0.0000,1.0000
C01251=117.270,43.250,10.200,-0.0000,-0.0000,1.0000
C01252=118.440,39.840,10.190,-0.0100,-0.0000,1.0000
C01253=119.490,36.210,10.190,-0.0200,-0.0100,1.0000
C01254=120.310,32.810,10.190,-0.0500,-0.0100,1.0000
C01255=120.820,30.090,10.180,-0.0900,-0.0100,1.0000
C01256=121.120,27.910,10.170,-0.1300,-0.0200,0.9900
C01257=121.380,25.750,10.140,-0.1700,-0.0200,0.9900
C01258=121.730,23.090,10.120,-0.2000,-0.0300,0.9800
C01259=122.270,19.220,10.100,-0.2300,-0.0300,0.9700
C01260=122.980,13.540,10.100,-0.2400,-0.0300,0.9700
C01261=123.520,7.120,10.100,-0.2400,-0.0100,0.9700
C01262=123.720,0.000,10.100,-0.2400,0.0000,0.9700
C01263=123.520,-7.120,10.100,-0.2400,0.0100,0.9700
C01264=122.980,-13.540,10.100,-0.2400,0.0300,0.9700
C01265=122.270,-19.220,10.100,-0.2300,0.0300,0.9700
C01266=121.730,-23.090,10.120,-0.2000,0.0300,0.9800
C01267=121.380,-25.750,10.140,-0.1700,0.0200,0.9900
C01268=121.120,-27.910,10.170,-0.1300,0.0200,0.9900
C01269=120.820,-30.090,10.180,-0.0900,0.0100,1.0000
C01270=120.310,-32.810,10.190,-0.0500,0.0100,1.0000
C01271=119.490,-36.210,10.190,-0.0200,0.0100,1.0000
C01272=118.440,-39.840,10.190,-0.0100,0.0000,1.0000
C01273=117.270,-43.250,10.200,-0.0000,0.0000,1.0000
C01274=116.090,-46.340,10.200,-0.0000,0.0000,1.0000
C01275=114.860,-49.320,10.200,-0.0000,0.0000,1.0000
C01276=113.510,-52.340,10.200,-0.0000,0.0000,1.0000
C01277=111.920,-55.580,10.190,-0.0100,0.0000,1.0000
C01278=110.100,-58.890,10.190,-0.0200,0.0100,1.0000
C01279=108.270,-61.870,10.190,-0.0400,0.0300,1.0000
C01280=106.710,-64.160,10.180,-0.0700,0.0500,1.0000
C01281=105.380,-65.910,10.170,-0.1000,0.0800,0.9900
C01282=104.040,-67.620,10.140,-0.1300,0.1100,0.9900
C01283=102.400,-69.750,10.120,-0.1600,0.1200,0.9800
C01284=100.050,-72.870,10.100,-0.1800,0.1400,0.9700
C01285=96.540,-77.390,10.100,-0.1900,0.1500,0.9700
C01286=92.380,-82.300,10.100,-0.1800,0.1600,0.9700
C01287=87.490,-87.490,10.100,-0.1700,0.1700,0.9700
C01288=82.300,-92.380,10.100,-0.1600,0.1800,0.9700
C01289=77.390,-96.540,10.100,-0.1500,0.1900,0.9700
C01290=72.870,-100.050,10.100,-0.1400,0.1800,0.9700
C01291=69.750,-102.400,10.120,-0.1200,0.1600,0.9800
C01292=67.620,-104.040,10.140,-0.1100,0.1300,0.9900
C01293=65.910,-105.380,10.170,-0.0800,0.1000,0.9900
C01294=64.160,-106.710,10.180,-0.0500,0.0700,1.0000
C01295=61.870,-108.270,10.190,-0.0300,0.0400,1.0000
C01296=58.890,-110.100,10.190,-0.0100,0.0200,1.0000
C01297=55.580,-111.920,10.190,-0.0000,0.0100,1.0000
C01298=52.340,-113.510,10.200,-0.0000,0.0000,1.0000
C01299=49.320,-114.860,10.200,-0.0000,0.0000,1.0000
C01300=46.340,-116.090,10.200,-0.0000,0.0000,1.0000
C01301=43.250,-117.270,10.200,-0.0000,0.0000,1.0000
C01302=39.840,-118.440,10.190,-0.0000,0.0100,1.0000
C01303=36.210,-119.490,10.190,-0.0100,0.0200,1.0000
C01304=32.810,-120.310,10.190,-0.0100,0.0500,1.0000
C01305=30.090,-120.820,10.180,-0.0100,0.0900,1.0000
C01306=27.910,-121.120,10.170,-0.0200,0.1300,0.9900
C01307=25.750,-121.380,10.140,-0.0200,0.1700,0.9900
C01308=23.090,-121.730,10.120,-0.0300,0.2000,0.9800
C01309=19.220,-122.270,10.100,-0.0300,0.2300,0.9700
C01310=13.540,-122.980,10.100,-0.0300,0.2400,0.9700
C01311=7.120,-123.520,10.100,-0.0100,0.2400,0.9700
C01312=0.000,-123.720,10.100,0.0000,0.2400,0.9700
C01313=0.000,-123.720,10.100,0.0000,0.2400,0.9700
C01314=-7.120,-123.520,10.100,0.0100,0.2400,0.9700
C01315=-13.540,-122.980,10.100,0.0300,0.2400,0.9700
C01316=-19.220,-122.270,10.100,0.0300,0.2300,0.9700
C01317=-23.090,-121.730,10.120,0.0300,0.2000,0.9800
C01318=-25.750,-121.380,10.140,0.0200,0.1700,0.9900
C01319=-27.910,-121.120,10.170,0.0200,0.1300,0.9900
C01320=-30.090,-120.820,10.180,0.0100,0.0900,1.0000
C01321=-32.810,-120.310,10.190,0.0100,0.0500,1.0000
C01322=-36.210,-119.490,10.190,0.0100,0.0200,1.0000
C01323=-39.840,-118.440,10.190,0.0000,0.0100,1.0000
C01324=-43.250,-117.270,10.200,0.0000,0.0000,1.0000
C01325=-46.340,-116.090,10.200,0.0000,0.0000,1.0000
C01326=-49.320,-114.860,10.200,0.0000,0.0000,1.0000
C01327=-52.340,-113.510,10.200,0.0000,0.0000,1.0000
C01328=-55.580,-111.920,10.190,0.0000,0.0100,1.0000
C01329=-58.890,-110.100,10.190,0.0100,0.0200,1.0000
C01330=-61.870,-108.270,10.190,0.0300,0.0400,1.0000
C01331=-64.160,-106.710,10.180,0.0500,0.0700,1.0000
C01332=-65.910,-105.380,10.170,0.0800,0.1000,0.9900
C01333=-67.620,-104.040,10.140,0.1100,0.1300,0.9900
C01334=-69.750,-102.400,10.120,0.1200,0.1600,0.9800
C01335=-72.870,-100.050,10.100,0.1400,0.1800,0.9700
C01336=-77.390,-96.540,10.100,0.1500,0.1900,0.9700
C01337=-82.300,-92.380,10.100,0.1600,0.1800,0.9700
C01338=-87.490,-87.490,10.100,0.1700,0.1700,0.9700
C01339=-92.380,-82.300,10.100,0.1800,0.1600,0.9700
C01340=-96.540,-77.390,10.100,0.1900,0.1500,0.9700
C01341=-100.050,-72.870,10.100,0.1800,0.1400,0.9700
C01342=-102.400,-69.750,10.120,0.1600,0.1200,0.9800
C01343=-104.040,-67.620,10.140,0.1300,0.1100,0.9900
C01344=-105.380,-65.910,10.170,0.1000,0.0800,0.9900
C01345=-106.710,-64.160,10.180,0.0700,0.0500,1.0000
C01346=-108.270,-61.870,10.190,0.0400,0.0300,1.0000
C01347=-110.100,-58.890,10.190,0.0200,0.0100,1.0000
C01348=-111.920,-55.580,10.190,0.0100,0.0000,1.0000
C01349=-113.510,-52.340,10.200,0.0000,0.0000,1.0000
C01350=-114.860,-49.320,10.200,0.0000,0.0000,1.0000
C01351=-116.090,-46.340,10.200,0.0000,0.0000,1.0000
C01352=-117.270,-43.250,10.200,0.0000,0.0000,1.0000
C01353=-118.440,-39.840,10.190,0.0100,0.0000,1.0000
C01354=-119.490,-36.210,10.190,0.0200,0.0100,1.0000
C01355=-120.310,-32.810,10.190,0.0500,0.0100,1.0000
C01356=-120.820,-30.090,10.180,0.0900,0.0100,1.0000
C01357=-121.120,-27.910,10.170,0.1300,0.0200,0.9900
C01358=-121.380,-25.750,10.140,0.1700,0.0200,0.9900
C01359=-121.730,-23.090,10.120,0.2000,0.0300,0.9800
C01360=-122.270,-19.220,10.100,0.2300,0.0300,0.9700
C01361=-122.980,-13.540,10.100,0.2400,0.0300,0.9700
C01362=-123.520,-7.120,10.100,0.2400,0.0100,0.9700
C01363=-123.720,0.000,10.100,0.2400,-0.0000,0.9700
C01364=-123.520,7.120,10.100,0.2400,-0.0100,0.9700
C01365=-122.980,13.540,10.100,0.2400,-0.0300,0.9700
C01366=-122.270,19.220,10.100,0.2300,-0.0300,0.9700
C01367=-121.730,23.090,10.120,0.2000,-0.0300,0.9800
C01368=-121.380,25.750,10.140,0.1700,-0.0200,0.9900
C01369=-121.120,27.910,10.170,0.1300,-0.0200,0.9900
C01370=-120.820,30.090,10.180,0.0900,-0.0100,1.0000
C01371=-120.310,32.810,10.190,0.0500,-0.0100,1.0000
C01372=-119.490,36.210,10.190,0.0200,-0.0100,1.0000
C01373=-118.440,39.840,10.190,0.0100,-0.0000,1.0000
C01374=-117.270,43.250,10.200,0.0000,-0.0000,1.0000
C01375=-116.090,46.340,10.200,0.0000,-0.0000,1.0000
C01376=-114.860,49.320,10.200,0.0000,-0.0000,1.0000
C01377=-113.510,52.340,10.200,0.0000,-0.0000,1.0000
C01378=-111.920,55.580,10.190,0.0100,-0.0000,1.0000
C01379=-110.100,58.890,10.190,0.0200,-0.0100,1.0000
C01380=-108.270,61.870,10.190,0.0400,-0.0300,1.0000
C01381=-106.710,64.160,10.180,0.0700,-0.0500,1.0000
C01382=-105.380,65.910,10.170,0.1000,-0.0800,0.9900
C01383=-104.040,67.620,10.140,0.1300,-0.1100,0.9900
C01384=-102.400,69.750,10.120,0.1600,-0.1200,0.9800
C01385=-100.050,72.870,10.100,0.1800,-0.1400,0.9700
C01386=-96.540,77.390,10.100,0.1900,-0.1500,0.9700
C01387=-92.380,82.300,10.100,0.1800,-0.1600,0.9700
C01388=-87.490,87.490,10.100,0.1700,-0.1700,0.9700
C01389=-82.300,92.380,10.100,0.1600,-0.1800,0.9700
C01390=-77.390,96.540,10.100,0.1500,-0.1900,0.9700
C01391=-72.870,100.050,10.100,0.1400,-0.1800,0.9700
C01392=-69.750,102.400,10.120,0.1200,-0.1600,0.9800
C01393=-67.620,104.040,10.140,0.1100,-0.1300,0.9900
C01394=-65.910,105.380,10.170,0.0800,-0.1000,0.9900
C01395=-64.160,106.710,10.180,0.0500,-0.0700,1.0000
C01396=-61.870,108.270,10.190,0.0300,-0.0400,1.0000
C01397=-58.890,110.100,10.190,0.0100,-0.0200,1.0000
C01398=-55.580,111.920,10.190,0.0000,-0.0100,1.0000
C01399=-52.340,113.510,10.200,0.0000,-0.0000,1.0000
C01400=-49.320,114.860,10.200,0.0000,-0.0000,1.0000
C01401=-46.340,116.090,10.200,0.0000,-0.0000,1.0000
C01402=-43.250,117.270,10.200,0.0000,-0.0000,1.0000
C01403=-39.840,118.440,10.190,0.0000,-0.0100,1.0000
C01404=-36.210,119.490,10.190,0.0100,-0.0200,1.0000
C01405=-32.810,120.310,10.190,0.0100,-0.0500,1.0000
C01406=-30.090,120.820,10.180,0.0100,-0.0900,1.0000
C01407=-27.910,121.120,10.170,0.0200,-0.1300,0.9900
C01408=-25.750,121.380,10.140,0.0200,-0.1700,0.9900
C01409=-23.090,121.730,10.120,0.0300,-0.2000,0.9800
C01410=-19.220,122.270,10.100,0.0300,-0.2300,0.9700
C01411=-13.540,122.980,10.100,0.0300,-0.2400,0.9700
C01412=-7.120,123.520,10.100,0.0100,-0.2400,0.9700
C01413=0.000,123.720,10.100,0.0000,-0.2400,0.9700
C01414=0.000,123.290,11.740,0.0000,-0.2700,0.9600
C01415=-7.080,123.080,11.740,0.0200,-0.2700,0.9600
C01416=-13.470,122.550,11.740,0.0300,-0.2700,0.9600
C01417=-19.140,121.860,11.750,0.0300,-0.2600,0.9700
C01418=-22.990,121.360,11.780,0.0300,-0.2300,0.9700
C01419=-25.640,121.070,11.810,0.0200,-0.1900,0.9800
C01420=-27.800,120.900,11.850,0.0100,-0.1500,0.9900
C01421=-29.970,120.680,11.870,0.0100,-0.1000,1.0000
C01422=-32.680,120.240,11.880,0.0100,-0.0600,1.0000
C01423=-36.090,119.480,11.890,0.0100,-0.0300,1.0000
C01424=-39.740,118.460,11.890,0.0000,-0.0100,1.0000
C01425=-43.190,117.290,11.900,0.0000,-0.0000,1.0000
C01426=-46.320,116.100,11.900,0.0000,-0.0000,1.0000
C01427=-49.340,114.850,11.900,0.0000,-0.0000,1.0000
C01428=-52.400,113.480,11.900,0.0000,-0.0000,1.0000
C01429=-55.660,111.860,11.890,0.0000,-0.0100,1.0000
C01430=-58.970,110.000,11.890,0.0100,-0.0200,1.0000
C01431=-61.910,108.130,11.880,0.0300,-0.0500,1.0000
C01432=-64.140,106.520,11.870,0.0600,-0.0800,1.0000
C01433=-65.830,105.140,11.850,0.0900,-0.1100,0.9900
C01434=-67.480,103.750,11.810,0.1200,-0.1500,0.9800
C01435=-69.560,102.070,11.780,0.1500,-0.1800,0.9700
C01436=-72.640,99.700,11.750,0.1600,-0.2100,0.9700
C01437=-77.130,96.180,11.740,0.1700,-0.2100,0.9600
C01438=-82.020,92.040,11.740,0.1800,-0.2000,0.9600
C01439=-87.180,87.180,11.740,0.1900,-0.1900,0.9600
C01440=-92.040,82.020,11.740,0.2000,-0.1800,0.9600
C01441=-96.180,77.130,11.740,0.2100,-0.1700,0.9600
C01442=-99.700,72.640,11.750,0.2100,-0.1600,0.9700
C01443=-102.070,69.560,11.780,0.1800,-0.1500,0.9700
C01444=-103.750,67.480,11.810,0.1500,-0.1200,0.9800
C01445=-105.140,65.830,11.850,0.1100,-0.0900,0.9900
C01446=-106.520,64.140,11.870,0.0800,-0.0600,1.0000
C01447=-108.130,61.910,11.880,0.0500,-0.0300,1.0000
C01448=-110.000,58.970,11.890,0.0200,-0.0100,1.0000
C01449=-111.860,55.660,11.890,0.0100,-0.0000,1.0000
C01450=-113.480,52.400,11.900,0.0000,-0.0000,1.0000
C01451=-114.850,49.340,11.900,0.0000,-0.0000,1.0000
C01452=-116.100,46.320,11.900,0.0000,-0.0000,1.0000
C01453=-117.290,43.190,11.900,0.0000,-0.0000,1.0000
C01454=-118.460,39.740,11.890,0.0100,-0.0000,1.0000
C01455=-119.480,36.090,11.890,0.0300,-0.0100,1.0000
C01456=-120.240,32.680,11.880,0.0600,-0.0100,1.0000
C01457=-120.680,29.970,11.870,0.1000,-0.0100,1.0000
C01458=-120.900,27.800,11.850,0.1500,-0.0100,0.9900
C01459=-121.070,25.640,11.810,0.1900,-0.0200,0.9800
C01460=-121.360,22.990,11.780,0.2300,-0.0300,0.9700
C01461=-121.860,19.140,11.750,0.2600,-0.0300,0.9700
C01462=-122.550,13.470,11.740,0.2700,-0.0300,0.9600
C01463=-123.080,7.080,11.740,0.2700,-0.0200,0.9600
C01464=-123.290,0.000,11.740,0.2700,-0.0000,0.9600
C01465=-123.080,-7.080,11.740,0.2700,0.0200,0.9600
C01466=-122.550,-13.470,11.740,0.2700,0.0300,0.9600
C01467=-121.860,-19.140,11.750,0.2600,0.0300,0.9700
C01468=-121.360,-22.990,11.780,0.2300,0.0300,0.9700
C01469=-121.070,-25.640,11.810,0.1900,0.0200,0.9800
C01470=-120.900,-27.800,11.850,0.1500,0.0100,0.9900
C01471=-120.680,-29.970,11.870,0.1000,0.0100,1.0000
C01472=-120.240,-32.680,11.880,0.0600,0.0100,1.0000
C01473=-119.480,-36.090,11.890,0.0300,0.0100,1.0000
C01474=-118.460,-39.740,11.890,0.0100,0.0000,1.0000
C01475=-117.290,-43.190,11.900,0.0000,0.0000,1.0000
C01476=-116.100,-46.320,11.900,0.0000,0.0000,1.0000
C01477=-114.850,-49.340,11.900,0.0000,0.0000,1.0000
C01478=-113.480,-52.400,11.900,0.0000,0.0000,1.0000
C01479=-111.860,-55.660,11.890,0.0100,0.0000,1.0000
C01480=-110.000,-58.970,11.890,0.0200,0.0100,1.0000
C01481=-108.130,-61.910,11.880,0.0500,0.0300,1.0000
C01482=-106.520,-64.140,11.870,0.0800,0.0600,1.0000
C01483=-105.140,-65.830,11.850,0.1100,0.0900,0.9900
C01484=-103.750,-67.480,11.810,0.1500,0.1200,0.9800
C01485=-102.070,-69.560,11.780,0.1800,0.1500,0.9700
C01486=-99.700,-72.640,11.750,0.2100,0.1600,0.9700
C01487=-96.180,-77.130,11.740,0.2100,0.1700,0.9600
C01488=-92.040,-82.020,11.740,0.2000,0.1800,0.9600
C01489=-87.180,-87.180,11.740,0.1900,0.1900,0.9600
C01490=-82.020,-92.040,11.740,0.1800,0.2000,0.9600
C01491=-77.130,-96.180,11.740,0.1700,0.2100,0.9600
C01492=-72.640,-99.700,11.750,0.1600,0.2100,0.9700
C01493=-69.560,-102.070,11.780,0.1500,0.1800,0.9700
C01494=-67.480,-103.750,11.810,0.1200,0.1500,0.9800
C01495=-65.830,-105.140,11.850,0.0900,0.1100,0.9900
C01496=-64.140,-106.520,11.870,0.0600,0.0800,1.0000
C01497=-61.910,-108.130,11.880,0.0300,0.0500,1.0000
C01498=-58.970,-110.000,11.890,0.0100,0.0200,1.0000
C01499=-55.660,-111.860,11.890,0.0000,0.0100,1.0000
C01500=-52.400,-113.480,11.900,0.0000,0.0000,1.0000
C01501=-49.340,-114.850,11.900,0.0000,0.0000,1.0000
C01502=-46.320,-116.100,11.900,0.0000,0.0000,1.0000
C01503=-43.190,-117.290,11.900,0.0000,0.0000,1.0000
C01504=-39.740,-118.460,11.890,0.0000,0.0100,1.0000
C01505=-36.090,-119.480,11.890,0.0100,0.0300,1.0000
C01506=-32.680,-120.240,11.880,0.0100,0.0600,1.0000
C01507=-29.970,-120.680,11.870,0.0100,0.1000,1.0000
C01508=-27.800,-120.900,11.850,0.0100,0.1500,0.9900
C01509=-25.640,-121.070,11.810,0.0200,0.1900,0.9800
C01510=-22.990,-121.360,11.780,0.0300,0.2300,0.9700
C01511=-19.140,-121.860,11.750,0.0300,0.2600,0.9700
C01512=-13.470,-122.550,11.740,0.0300,0.2700,0.9600
C01513=-7.080,-123.080,11.740,0.0200,0.2700,0.9600
C01514=0.000,-123.290,11.740,0.0000,0.2700,0.9600
C01515=0.000,-123.290,11.740,0.0000,0.2700,0.9600
C01516=7.080,-123.080,11.740,-0.0200,0.2700,0.9600
C01517=13.470,-122.550,11.740,-0.0300,0.2700,0.9600
C01518=19.140,-121.860,11.750,-0.0300,0.2600,0.9700
C01519=22.990,-121.360,11.780,-0.0300,0.2300,0.9700
C01520=25.640,-121.070,11.810,-0.0200,0.1900,0.9800
C01521=27.800,-120.900,11.850,-0.0100,0.1500,0.9900
C01522=29.970,-120.680,11.870,-0.0100,0.1000,1.0000
C01523=32.680,-120.240,11.880,-0.0100,0.0600,1.0000
C01524=36.090,-119.480,11.890,-0.0100,0.0300,1.0000
C01525=39.740,-118.460,11.890,-0.0000,0.0100,1.0000
C01526=43.190,-117.290,11.900,-0.0000,0.0000,1.0000
C01527=46.320,-116.100,11.900,-0.0000,0.0000,1.0000
C01528=49.340,-114.850,11.900,-0.0000,0.0000,1.0000
C01529=52.400,-113.480,11.900,-0.0000,0.0000,1.0000
C01530=55.660,-111.860,11.890,-0.0000,0.0100,1.0000
C01531=58.970,-110.000,11.890,-0.0100,0.0200,1.0000
C01532=61.910,-108.130,11.880,-0.0300,0.0500,1.0000
C01533=64.140,-106.520,11.870,-0.0600,0.0800,1.0000
C01534=65.830,-105.140,11.850,-0.0900,0.1100,0.9900
C01535=67.480,-103.750,11.810,-0.1200,0.1500,0.9800
C01536=69.560,-102.070,11.780,-0.1500,0.1800,0.9700
C01537=72.640,-99.700,11.750,-0.1600,0.2100,0.9700
C01538=77.130,-96.180,11.740,-0.1700,0.2100,0.9600
C01539=82.020,-92.040,11.740,-0.1800,0.2000,0.9600
C01540=87.180,-87.180,11.740,-0.1900,0.1900,0.9600
C01541=92.040,-82.020,11.740,-0.2000,0.1800,0.9600
C01542=96.180,-77.130,11.740,-0.2100,0.1700,0.9600
C01543=99.700,-72.640,11.750,-0.2100,0.1600,0.9700
C01544=102.070,-69.560,11.780,-0.1800,0.1500,0.9700
C01545=103.750,-67.480,11.810,-0.1500,0.1200,0.9800
C01546=105.140,-65.830,11.850,-0.1100,0.0900,0.9900
C01547=106.520,-64.140,11.870,-0.0800,0.0600,1.0000
C01548=108.130,-61.910,11.880,-0.0500,0.0300,1.0000
C01549=110.000,-58.970,11.890,-0.0200,0.0100,1.0000
C01550=111.860,-55.660,11.890,-0.0100,0.0000,1.0000
C01551=113.480,-52.400,11.900,-0.0000,0.0000,1.0000
C01552=114.850,-49.340,11.900,-0.0000,0.0000,1.0000
C01553=116.100,-46.320,11.900,-0.0000,0.0000,1.0000
C01554=117.290,-43.190,11.900,-0.0000,0.0000,1.0000
C01555=118.460,-39.740,11.890,-0.0100,0.0000,1.0000
C01556=119.480,-36.090,11.890,-0.0300,0.0100,1.0000
C01557=120.240,-32.680,11.880,-0.0600,0.0100,1.0000
C01558=120.680,-29.970,11.870,-0.1000,0.0100,1.0000
C01559=120.900,-27.800,11.850,-0.1500,0.0100,0.9900
C01560=121.070,-25.640,11.810,-0.1900,0.0200,0.9800
C01561=121.360,-22.990,11.780,-0.2300,0.0300,0.9700
C01562=121.860,-19.140,11.750,-0.2600,0.0300,0.9700
C01563=122.550,-13.470,11.740,-0.2700,0.0300,0.9600
C01564=123.080,-7.080,11.740,-0.2700,0.0200,0.9600
C01565=123.290,0.000,11.740,-0.2700,0.0000,0.9600
C01566=123.080,7.080,11.740,-0.2700,-0.0200,0.9600
C01567=122.550,13.470,11.740,-0.2700,-0.0300,0.9600
C01568=121.860,19.140,11.750,-0.2600,-0.0300,0.9700
C01569=121.360,22.990,11.780,-0.2300,-0.0300,0.9700
C01570=121.070,25.640,11.810,-0.1900,-0.0200,0.9800
C01571=120.900,27.800,11.850,-0.1500,-0.0100,0.9900
C01572=120.680,29.970,11.870,-0.1000,-0.0100,1.0000
C01573=120.240,32.680,11.880,-0.0600,-0.0100,1.0000
C01574=119.480,36.090,11.890,-0.0300,-0.0100,1.0000
C01575=118.460,39.740,11.890,-0.0100,-0.0000,1.0000
C01576=117.290,43.190,11.900,-0.0000,-0.0000,1.0000
C01577=116.100,46.320,11.900,-0.0000,-0.0000,1.0000
C01578=114.850,49.340,11.900,-0.0000,-0.0000,1.0000
C01579=113.480,52.400,11.900,-0.0000,-0.0000,1.0000
C01580=111.860,55.660,11.890,-0.0100,-0.0000,1.0000
C01581=110.000,58.970,11.890,-0.0200,-0.0100,1.0000
C01582=108.130,61.910,11.880,-0.0500,-0.0300,1.0000
C01583=106.520,64.140,11.870,-0.0800,-0.0600,1.0000
C01584=105.140,65.830,11.850,-0.1100,-0.0900,0.9900
C01585=103.750,67.480,11.810,-0.1500,-0.1200,0.9800
C01586=102.070,69.560,11.780,-0.1800,-0.1500,0.9700
C01587=99.700,72.640,11.750,-0.2100,-0.1600,0.9700
C01588=96.180,77.130,11.740,-0.2100,-0.1700,0.9600
C01589=92.040,82.020,11.740,-0.2000,-0.1800,0.9600
C01590=87.180,87.180,11.740,-0.1900,-0.1900,0.9600
C01591=82.020,92.040,11.740,-0.1800,-0.2000,0.9600
C01592=77.130,96.180,11.740,-0.1700,-0.2100,0.9600
C01593=72.640,99.700,11.750,-0.1600,-0.2100,0.9700
C01594=69.560,102.070,11.780,-0.1500,-0.1800,0.9700
C01595=67.480,103.750,11.810,-0.1200,-0.1500,0.9800
C01596=65.830,105.140,11.850,-0.0900,-0.1100,0.9900
C01597=64.140,106.520,11.870,-0.0600,-0.0800,1.0000
C01598=61.910,108.130,11.880,-0.0300,-0.0500,1.0000
C01599=58.970,110.000,11.890,-0.0100,-0.0200,1.0000
C01600=55.660,111.860,11.890,-0.0000,-0.0100,1.0000
C01601=52.400,113.480,11.900,-0.0000,-0.0000,1.0000
C01602=49.340,114.850,11.900,-0.0000,-0.0000,1.0000
C01603=46.320,116.100,11.900,-0.0000,-0.0000,1.0000
C01604=43.190,117.290,11.900,-0.0000,-0.0000,1.0000
C01605=39.740,118.460,11.890,-0.0000,-0.0100,1.0000
C01606=36.090,119.480,11.890,-0.0100,-0.0300,1.0000
C01607=32.680,120.240,11.880,-0.0100,-0.0600,1.0000
C01608=29.970,120.680,11.870,-0.0100,-0.1000,1.0000
C01609=27.800,120.900,11.850,-0.0100,-0.1500,0.9900
C01610=25.640,121.070,11.810,-0.0200,-0.1900,0.9800
C01611=22.990,121.360,11.780,-0.0300,-0.2300,0.9700
C01612=19.140,121.860,11.750,-0.0300,-0.2600,0.9700
C01613=13.470,122.550,11.740,-0.0300,-0.2700,0.9600
C01614=7.080,123.080,11.740,-0.0200,-0.2700,0.9600
C01615=0.000,123.290,11.740,0.0000,-0.2700,0.9600
C01616=0.000,122.800,13.370,0.0000,-0.3000,0.9500
C01617=7.040,122.600,13.370,-0.0200,-0.3000,0.9500
C01618=13.400,122.070,13.370,-0.0300,-0.3000,0.9500
C01619=19.040,121.400,13.380,-0.0400,-0.2900,0.9600
C01620=22.880,120.950,13.420,-0.0300,-0.2600,0.9700
C01621=25.520,120.740,13.480,-0.0100,-0.2100,0.9800
C01622=27.670,120.640,13.520,-0.0100,-0.1600,0.9900
C01623=29.830,120.520,13.560,-0.0100,-0.1100,0.9900
C01624=32.530,120.160,13.570,-0.0100,-0.0600,1.0000
C01625=35.950,119.460,13.580,-0.0100,-0.0300,1.0000
C01626=39.630,118.480,13.590,-0.0000,-0.0100,1.0000
C01627=43.120,117.320,13.600,-0.0000,-0.0000,1.0000
C01628=46.300,116.110,13.600,-0.0000,-0.0000,1.0000
C01629=49.360,114.840,13.600,-0.0000,-0.0000,1.0000
C01630=52.460,113.440,13.600,-0.0000,-0.0000,1.0000
C01631=55.750,111.800,13.590,-0.0000,-0.0100,1.0000
C01632=59.050,109.890,13.580,-0.0200,-0.0300,1.0000
C01633=61.960,107.970,13.570,-0.0400,-0.0500,1.0000
C01634=64.120,106.310,13.560,-0.0700,-0.0800,0.9900
C01635=65.740,104.870,13.520,-0.1100,-0.1200,0.9900
C01636=67.330,103.420,13.480,-0.1400,-0.1600,0.9800
C01637=69.340,101.700,13.420,-0.1700,-0.2000,0.9700
C01638=72.380,99.310,13.380,-0.1800,-0.2300,0.9600
C01639=76.840,95.790,13.370,-0.1900,-0.2300,0.9500
C01640=81.710,91.670,13.370,-0.2000,-0.2300,0.9500
C01641=86.830,86.830,13.370,-0.2100,-0.2100,0.9500
C01642=91.670,81.710,13.370,-0.2300,-0.2000,0.9500
C01643=95.790,76.840,13.370,-0.2300,-0.1900,0.9500
C01644=99.310,72.380,13.380,-0.2300,-0.1800,0.9600
C01645=101.700,69.340,13.420,-0.2000,-0.1700,0.9700
C01646=103.420,67.330,13.480,-0.1600,-0.1400,0.9800
C01647=104.870,65.740,13.520,-0.1200,-0.1100,0.9900
C01648=106.310,64.120,13.560,-0.0800,-0.0700,0.9900
C01649=107.970,61.960,13.570,-0.0500,-0.0400,1.0000
C01650=109.890,59.050,13.580,-0.0300,-0.0200,1.0000
C01651=111.800,55.750,13.590,-0.0100,-0.0000,1.0000
C01652=113.440,52.460,13.600,-0.0000,-0.0000,1.0000
C01653=114.840,49.360,13.600,-0.0000,-0.0000,1.0000
C01654=116.110,46.300,13.600,-0.0000,-0.0000,1.0000
C01655=117.320,43.120,13.600,-0.0000,-0.0000,1.0000
C01656=118.480,39.630,13.590,-0.0100,-0.0000,1.0000
C01657=119.460,35.950,13.580,-0.0300,-0.0100,1.0000
C01658=120.160,32.530,13.570,-0.0600,-0.0100,1.0000
C01659=120.520,29.830,13.560,-0.1100,-0.0100,0.9900
C01660=120.640,27.670,13.520,-0.1600,-0.0100,0.9900
C01661=120.740,25.520,13.480,-0.2100,-0.0100,0.9800
C01662=120.950,22.880,13.420,-0.2600,-0.0300,0.9700
C01663=121.400,19.040,13.380,-0.2900,-0.0400,0.9600
C01664=122.070,13.400,13.370,-0.3000,-0.0300,0.9500
C01665=122.600,7.040,13.370,-0.3000,-0.0200,0.9500
C01666=122.800,0.000,13.370,-0.3000,0.0000,0.9500
C01667=122.600,-7.040,13.370,-0.3000,0.0200,0.9500
C01668=122.070,-13.400,13.370,-0.3000,0.0300,0.9500
C01669=121.400,-19.040,13.380,-0.2900,0.0400,0.9600
C01670=120.950,-22.880,13.420,-0.2600,0.0300,0.9700
C01671=120.740,-25.520,13.480,-0.2100,0.0100,0.9800
C01672=120.640,-27.670,13.520,-0.1600,0.0100,0.9900
C01673=120.520,-29.830,13.560,-0.1100,0.0100,0.9900
C01674=120.160,-32.530,13.570,-0.0600,0.0100,1.0000
C01675=119.460,-35.950,13.580,-0.0300,0.0100,1.0000
C01676=118.480,-39.630,13.590,-0.0100,0.0000,1.0000
C01677=117.320,-43.120,13.600,-0.0000,0.0000,1.0000
C01678=116.110,-46.300,13.600,-0.0000,0.0000,1.0000
C01679=114.840,-49.360,13.600,-0.0000,0.0000,1.0000
C01680=113.440,-52.460,13.600,-0.0000,0.0000,1.0000
C01681=111.800,-55.750,13.590,-0.0100,0.0000,1.0000
C01682=109.890,-59.050,13.580,-0.0300,0.0200,1.0000
C01683=107.970,-61.960,13.570,-0.0500,0.0400,1.0000
C01684=106.310,-64.120,13.560,-0.0800,0.0700,0.9900
C01685=104.870,-65.740,13.520,-0.1200,0.1100,0.9900
C01686=103.420,-67.330,13.480,-0.1600,0.1400,0.9800
C01687=101.700,-69.340,13.420,-0.2000,0.1700,0.9700
C01688=99.310,-72.380,13.380,-0.2300,0.1800,0.9600
C01689=95.790,-76.840,13.370,-0.2300,0.1900,0.9500
C01690=91.670,-81.710,13.370,-0.2300,0.2000,0.9500
C01691=86.830,-86.830,13.370,-0.2100,0.2100,0.9500
C01692=81.710,-91.670,13.370,-0.2000,0.2300,0.9500
C01693=76.840,-95.790,13.370,-0.1900,0.2300,0.9500
C01694=72.380,-99.310,13.380,-0.1800,0.2300,0.9600
C01695=69.340,-101.700,13.420,-0.1700,0.2000,0.9700
C01696=67.330,-103.420,13.480,-0.1400,0.1600,0.9800
C01697=65.740,-104.870,13.520,-0.1100,0.1200,0.9900
C01698=64.120,-106.310,13.560,-0.0700,0.0800,0.9900
C01699=61.960,-107.970,13.570,-0.0400,0.0500,1.0000
C01700=59.050,-109.890,13.580,-0.0200,0.0300,1.0000
C01701=55.750,-111.800,13.590,-0.0000,0.0100,1.0000
C01702=52.460,-113.440,13.600,-0.0000,0.0000,1.0000
C01703=49.360,-114.840,13.600,-0.0000,0.0000,1.0000
C01704=46.300,-116.110,13.600,-0.0000,0.0000,1.0000
C01705=43.120,-117.320,13.600,-0.0000,0.0000,1.0000
C01706=39.630,-118.480,13.590,-0.0000,0.0100,1.0000
C01707=35.950,-119.460,13.580,-0.0100,0.0300,1.0000
C01708=32.530,-120.160,13.570,-0.0100,0.0600,1.0000
C01709=29.830,-120.520,13.560,-0.0100,0.1100,0.9900
C01710=27.670,-120.640,13.520,-0.0100,0.1600,0.9900
C01711=25.520,-120.740,13.480,-0.0100,0.2100,0.9800
C01712=22.880,-120.950,13.420,-0.0300,0.2600,0.9700
C01713=19.040,-121.400,13.380,-0.0400,0.2900,0.9600
C01714=13.400,-122.070,13.370,-0.0300,0.3000,0.9500
C01715=7.040,-122.600,13.370,-0.0200,0.3000,0.9500
C01716=0.000,-122.800,13.370,0.0000,0.3000,0.9500
C01717=0.000,-122.800,13.370,0.0000,0.3000,0.9500
C01718=-7.040,-122.600,13.370,0.0200,0.3000,0.9500
C01719=-13.400,-122.070,13.370,0.0300,0.3000,0.9500
C01720=-19.040,-121.400,13.380,0.0400,0.2900,0.9600
C01721=-22.880,-120.950,13.420,0.0300,0.2600,0.9700
C01722=-25.520,-120.740,13.480,0.0100,0.2100,0.9800
C01723=-27.670,-120.640,13.520,0.0100,0.1600,0.9900
C01724=-29.830,-120.520,13.560,0.0100,0.1100,0.9900
C01725=-32.530,-120.160,13.570,0.0100,0.0600,1.0000
C01726=-35.950,-119.460,13.580,0.0100,0.0300,1.0000
C01727=-39.630,-118.480,13.590,0.0000,0.0100,1.0000
C01728=-43.120,-117.320,13.600,0.0000,0.0000,1.0000
C01729=-46.300,-116.110,13.600,0.0000,0.0000,1.0000
C01730=-49.360,-114.840,13.600,0.0000,0.0000,1.0000
C01731=-52.460,-113.440,13.600,0.0000,0.0000,1.0000
C01732=-55.750,-111.800,13.590,0.0000,0.0100,1.0000
C01733=-59.050,-109.890,13.580,0.0200,0.0300,1.0000
C01734=-61.960,-107.970,13.570,0.0400,0.0500,1.0000
C01735=-64.120,-106.310,13.560,0.0700,0.0800,0.9900
C01736=-65.740,-104.870,13.520,0.1100,0.1200,0.9900
C01737=-67.330,-103.420,13.480,0.1400,0.1600,0.9800
C01738=-69.340,-101.700,13.420,0.1700,0.2000,0.9700
C01739=-72.380,-99.310,13.380,0.1800,0.2300,0.9600
C01740=-76.840,-95.790,13.370,0.1900,0.2300,0.9500
C01741=-81.710,-91.670,13.370,0.2000,0.2300,0.9500
C01742=-86.830,-86.830,13.370,0.2100,0.2100,0.9500
C01743=-91.670,-81.710,13.370,0.2300,0.2000,0.9500
C01744=-95.790,-76.840,13.370,0.2300,0.1900,0.9500
C01745=-99.310,-72.380,13.380,0.2300,0.1800,0.9600
C01746=-101.700,-69.340,13.420,0.2000,0.1700,0.9700
C01747=-103.420,-67.330,13.480,0.1600,0.1400,0.9800
C01748=-104.870,-65.740,13.520,0.1200,0.1100,0.9900
C01749=-106.310,-64.120,13.560,0.0800,0.0700,0.9900
C01750=-107.970,-61.960,13.570,0.0500,0.0400,1.0000
C01751=-109.890,-59.050,13.580,0.0300,0.0200,1.0000
C01752=-111.800,-55.750,13.590,0.0100,0.0000,1.0000
C01753=-113.440,-52.460,13.600,0.0000,0.0000,1.0000
C01754=-114.840,-49.360,13.600,0.0000,0.0000,1.0000
C01755=-116.110,-46.300,13.600,0.0000,0.0000,1.0000
C01756=-117.320,-43.120,13.600,0.0000,0.0000,1.0000
C01757=-118.480,-39.630,13.590,0.0100,0.0000,1.0000
C01758=-119.460,-35.950,13.580,0.0300,0.0100,1.0000
C01759=-120.160,-32.530,13.570,0.0600,0.0100,1.0000
C01760=-120.520,-29.830,13.560,0.1100,0.0100,0.9900
C01761=-120.640,-27.670,13.520,0.1600,0.0100,0.9900
C01762=-120.740,-25.520,13.480,0.2100,0.0100,0.9800
C01763=-120.950,-22.880,13.420,0.2600,0.0300,0.9700
C01764=-121.400,-19.040,13.380,0.2900,0.0400,0.9600
C01765=-122.070,-13.400,13.370,0.3000,0.0300,0.9500
C01766=-122.600,-7.040,13.370,0.3000,0.0200,0.9500
C01767=-122.800,0.000,13.370,0.3000,-0.0000,0.9500
C01768=-122.600,7.040,13.370,0.3000,-0.0200,0.9500
C01769=-122.070,13.400,13.370,0.3000,-0.0300,0.9500
C01770=-121.400,19.040,13.380,0.2900,-0.0400,0.9600
C01771=-120.950,22.880,13.420,0.2600,-0.0300,0.9700
C01772=-120.740,25.520,13.480,0.2100,-0.0100,0.9800
C01773=-120.640,27.670,13.520,0.1600,-0.0100,0.9900
C01774=-120.520,29.830,13.560,0.1100,-0.0100,0.9900
C01775=-120.160,32.530,13.570,0.0600,-0.0100,1.0000
C01776=-119.460,35.950,13.580,0.0300,-0.0100,1.0000
C01777=-118.480,39.630,13.590,0.0100,-0.0000,1.0000
C01778=-117.320,43.120,13.600,0.0000,-0.0000,1.0000
C01779=-116.110,46.300,13.600,0.0000,-0.0000,1.0000
C01780=-114.840,49.360,13.600,0.0000,-0.0000,1.0000
C01781=-113.440,52.460,13.600,0.0000,-0.0000,1.0000
C01782=-111.800,55.750,13.590,0.0100,-0.0000,1.0000
C01783=-109.890,59.050,13.580,0.0300,-0.0200,1.0000
C01784=-107.970,61.960,13.570,0.0500,-0.0400,1.0000
C01785=-106.310,64.120,13.560,0.0800,-0.0700,0.9900
C01786=-104.870,65.740,13.520,0.1200,-0.1100,0.9900
C01787=-103.420,67.330,13.480,0.1600,-0.1400,0.9800
C01788=-101.700,69.340,13.420,0.2000,-0.1700,0.9700
C01789=-99.310,72.380,13.380,0.2300,-0.1800,0.9600
C01790=-95.790,76.840,13.370,0.2300,-0.1900,0.9500
C01791=-91.670,81.710,13.370,0.2300,-0.2000,0.9500
C01792=-86.830,86.830,13.370,0.2100,-0.2100,0.9500
C01793=-81.710,91.670,13.370,0.2000,-0.2300,0.9500
C01794=-76.840,95.790,13.370,0.1900,-0.2300,0.9500
C01795=-72.380,99.310,13.380,0.1800,-0.2300,0.9600
C01796=-69.340,101.700,13.420,0.1700,-0.2000,0.9700
C01797=-67.330,103.420,13.480,0.1400,-0.1600,0.9800
C01798=-65.740,104.870,13.520,0.1100,-0.1200,0.9900
C01799=-64.120,106.310,13.560,0.0700,-0.0800,0.9900
C01800=-61.960,107.970,13.570,0.0400,-0.0500,1.0000
C01801=-59.050,109.890,13.580,0.0200,-0.0300,1.0000
C01802=-55.750,111.800,13.590,0.0000,-0.0100,1.0000
C01803=-52.460,113.440,13.600,0.0000,-0.0000,1.0000
C01804=-49.360,114.840,13.600,0.0000,-0.0000,1.0000
C01805=-46.300,116.110,13.600,0.0000,-0.0000,1.0000
C01806=-43.120,117.320,13.600,0.0000,-0.0000,1.0000
C01807=-39.630,118.480,13.590,0.0000,-0.0100,1.0000
C01808=-35.950,119.460,13.580,0.0100,-0.0300,1.0000
C01809=-32.530,120.160,13.570,0.0100,-0.0600,1.0000
C01810=-29.830,120.520,13.560,0.0100,-0.1100,0.9900
C01811=-27.670,120.640,13.520,0.0100,-0.1600,0.9900
C01812=-25.520,120.740,13.480,0.0100,-0.2100,0.9800
C01813=-22.880,120.950,13.420,0.0300,-0.2600,0.9700
C01814=-19.040,121.400,13.380,0.0400,-0.2900,0.9600
C01815=-13.400,122.070,13.370,0.0300,-0.3000,0.9500
C01816=-7.040,122.600,13.370,0.0200,-0.3000,0.9500
C01817=0.000,122.800,13.370,0.0000,-0.3000,0.9500
C01818=0.000,122.260,14.980,0.0000,-0.3300,0.9400
C01819=-6.990,122.060,14.980,0.0200,-0.3300,0.9400
C01820=-13.310,121.540,14.980,0.0300,-0.3300,0.9400
C01821=-18.940,120.890,15.000,0.0400,-0.3200,0.9500
C01822=-22.760,120.490,15.060,0.0200,-0.2800,0.9600
C01823=-25.390,120.360,15.130,0.0000,-0.2300,0.9700
C01824=-27.520,120.360,15.190,-0.0000,-0.1700,0.9800
C01825=-29.680,120.330,15.240,0.0100,-0.1200,0.9900
C01826=-32.370,120.070,15.260,0.0100,-0.0700,1.0000
C01827=-35.790,119.440,15.270,0.0100,-0.0300,1.0000
C01828=-39.510,118.500,15.280,0.0000,-0.0100,1.0000
C01829=-43.040,117.340,15.290,0.0000,-0.0000,1.0000
C01830=-46.270,116.120,15.300,0.0000,-0.0000,1.0000
C01831=-49.390,114.830,15.300,0.0000,-0.0000,1.0000
C01832=-52.540,113.410,15.290,0.0000,-0.0000,1.0000
C01833=-55.850,111.730,15.280,0.0000,-0.0100,1.0000
C01834=-59.150,109.770,15.270,0.0200,-0.0300,1.0000
C01835=-62.010,107.790,15.260,0.0400,-0.0600,1.0000
C01836=-64.100,106.080,15.240,0.0800,-0.0900,0.9900
C01837=-65.650,104.570,15.190,0.1200,-0.1200,0.9800
C01838=-67.150,103.060,15.130,0.1600,-0.1700,0.9700
C01839=-69.110,101.290,15.060,0.1900,-0.2200,0.9600
C01840=-72.090,98.880,15.000,0.2000,-0.2500,0.9500
C01841=-76.530,95.360,14.980,0.2100,-0.2600,0.9400
C01842=-81.370,91.250,14.980,0.2200,-0.2500,0.9400
C01843=-86.450,86.450,14.980,0.2300,-0.2300,0.9400
C01844=-91.250,81.370,14.980,0.2500,-0.2200,0.9400
C01845=-95.360,76.530,14.980,0.2600,-0.2100,0.9400
C01846=-98.880,72.090,15.000,0.2500,-0.2000,0.9500
C01847=-101.290,69.110,15.060,0.2200,-0.1900,0.9600
C01848=-103.060,67.150,15.130,0.1700,-0.1600,0.9700
C01849=-104.570,65.650,15.190,0.1200,-0.1200,0.9800
C01850=-106.080,64.100,15.240,0.0900,-0.0800,0.9900
C01851=-107.790,62.010,15.260,0.0600,-0.0400,1.0000
C01852=-109.770,59.150,15.270,0.0300,-0.0200,1.0000
C01853=-111.730,55.850,15.280,0.0100,-0.0000,1.0000
C01854=-113.410,52.540,15.290,0.0000,-0.0000,1.0000
C01855=-114.830,49.390,15.300,0.0000,-0.0000,1.0000
C01856=-116.120,46.270,15.300,0.0000,-0.0000,1.0000
C01857=-117.340,43.040,15.290,0.0000,-0.0000,1.0000
C01858=-118.500,39.510,15.280,0.0100,-0.0000,1.0000
C01859=-119.440,35.790,15.270,0.0300,-0.0100,1.0000
C01860=-120.070,32.370,15.260,0.0700,-0.0100,1.0000
C01861=-120.330,29.680,15.240,0.1200,-0.0100,0.9900
C01862=-120.360,27.520,15.190,0.1700,0.0000,0.9800
C01863=-120.360,25.390,15.130,0.2300,-0.0000,0.9700
C01864=-120.490,22.760,15.060,0.2800,-0.0200,0.9600
C01865=-120.890,18.940,15.000,0.3200,-0.0400,0.9500
C01866=-121.540,13.310,14.980,0.3300,-0.0300,0.9400
C01867=-122.060,6.990,14.980,0.3300,-0.0200,0.9400
C01868=-122.260,0.000,14.980,0.3300,-0.0000,0.9400
C01869=-122.060,-6.990,14.980,0.3300,0.0200,0.9400
C01870=-121.540,-13.310,14.980,0.3300,0.0300,0.9400
C01871=-120.890,-18.940,15.000,0.3200,0.0400,0.9500
C01872=-120.490,-22.760,15.060,0.2800,0.0200,0.9600
C01873=-120.360,-25.390,15.130,0.2300,0.0000,0.9700
C01874=-120.360,-27.520,15.190,0.1700,-0.0000,0.9800
C01875=-120.330,-29.680,15.240,0.1200,0.0100,0.9900
C01876=-120.070,-32.370,15.260,0.0700,0.0100,1.0000
C01877=-119.440,-35.790,15.270,0.0300,0.0100,1.0000
C01878=-118.500,-39.510,15.280,0.0100,0.0000,1.0000
C01879=-117.340,-43.040,15.290,0.0000,0.0000,1.0000
C01880=-116.120,-46.270,15.300,0.0000,0.0000,1.0000
C01881=-114.830,-49.390,15.300,0.0000,0.0000,1.0000
C01882=-113.410,-52.540,15.290,0.0000,0.0000,1.0000
C01883=-111.730,-55.850,15.280,0.0100,0.0000,1.0000
C01884=-109.770,-59.150,15.270,0.0300,0.0200,1.0000
C01885=-107.790,-62.010,15.260,0.0600,0.0400,1.0000
C01886=-106.080,-64.100,15.240,0.0900,0.0800,0.9900
C01887=-104.570,-65.650,15.190,0.1200,0.1200,0.9800
C01888=-103.060,-67.150,15.130,0.1700,0.1600,0.9700
C01889=-101.290,-69.110,15.060,0.2200,0.1900,0.9600
C01890=-98.880,-72.090,15.000,0.2500,0.2000,0.9500
C01891=-95.360,-76.530,14.980,0.2600,0.2100,0.9400
C01892=-91.250,-81.370,14.980,0.2500,0.2200,0.9400
C01893=-86.450,-86.450,14.980,0.2300,0.2300,0.9400
C01894=-81.370,-91.250,14.980,0.2200,0.2500,0.9400
C01895=-76.530,-95.360,14.980,0.2100,0.2600,0.9400
C01896=-72.090,-98.880,15.000,0.2000,0.2500,0.9500
C01897=-69.110,-101.290,15.060,0.1900,0.2200,0.9600
C01898=-67.150,-103.060,15.130,0.1600,0.1700,0.9700
C01899=-65.650,-104.570,15.190,0.1200,0.1200,0.9800
C01900=-64.100,-106.080,15.240,0.0800,0.0900,0.9900
C01901=-62.010,-107.790,15.260,0.0400,0.0600,1.0000
C01902=-59.150,-109.770,15.270,0.0200,0.0300,1.0000
C01903=-55.850,-111.730,15.280,0.0000,0.0100,1.0000
C01904=-52.540,-113.410,15.290,0.0000,0.0000,1.0000
C01905=-49.390,-114.830,15.300,0.0000,0.0000,1.0000
C01906=-46.270,-116.120,15.300,0.0000,0.0000,1.0000
C01907=-43.040,-117.340,15.290,0.0000,0.0000,1.0000
C01908=-39.510,-118.500,15.280,0.0000,0.0100,1.0000
C01909=-35.790,-119.440,15.270,0.0100,0.0300,1.0000
C01910=-32.370,-120.070,15.260,0.0100,0.0700,1.0000
C01911=-29.680,-120.330,15.240,0.0100,0.1200,0.9900
C01912=-27.520,-120.360,15.190,-0.0000,0.1700,0.9800
C01913=-25.390,-120.360,15.130,0.0000,0.2300,0.9700
C01914=-22.760,-120.490,15.060,0.0200,0.2800,0.9600
C01915=-18.940,-120.890,15.000,0.0400,0.3200,0.9500
C01916=-13.310,-121.540,14.980,0.0300,0.3300,0.9400
C01917=-6.990,-122.060,14.980,0.0200,0.3300,0.9400
C01918=0.000,-122.260,14.980,0.0000,0.3300,0.9400
C01919=0.000,-122.260,14.980,0.0000,0.3300,0.9400
C01920=6.990,-122.060,14.980,-0.0200,0.3300,0.9400
C01921=13.310,-121.540,14.980,-0.0300,0.3300,0.9400
C01922=18.940,-120.890,15.000,-0.0400,0.3200,0.9500
C01923=22.760,-120.490,15.060,-0.0200,0.2800,0.9600
C01924=25.390,-120.360,15.130,-0.0000,0.2300,0.9700
C01925=27.520,-120.360,15.190,0.0000,0.1700,0.9800
C01926=29.680,-120.330,15.240,-0.0100,0.1200,0.9900
C01927=32.370,-120.070,15.260,-0.0100,0.0700,1.0000
C01928=35.790,-119.440,15.270,-0.0100,0.0300,1.0000
C01929=39.510,-118.500,15.280,-0.0000,0.0100,1.0000
C01930=43.040,-117.340,15.290,-0.0000,0.0000,1.0000
C01931=46.270,-116.120,15.300,-0.0000,0.0000,1.0000
C01932=49.390,-114.830,15.300,-0.0000,0.0000,1.0000
C01933=52.540,-113.410,15.290,-0.0000,0.0000,1.0000
C01934=55.850,-111.730,15.280,-0.0000,0.0100,1.0000
C01935=59.150,-109.770,15.270,-0.0200,0.0300,1.0000
C01936=62.010,-107.790,15.260,-0.0400,0.0600,1.0000
C01937=64.100,-106.080,15.240,-0.0800,0.0900,0.9900
C01938=65.650,-104.570,15.190,-0.1200,0.1200,0.9800
C01939=67.150,-103.060,15.130,-0.1600,0.1700,0.9700
C01940=69.110,-101.290,15.060,-0.1900,0.2200,0.9600
C01941=72.090,-98.880,15.000,-0.2000,0.2500,0.9500
C01942=76.530,-95.360,14.980,-0.2100,0.2600,0.9400
C01943=81.370,-91.250,14.980,-0.2200,0.2500,0.9400
C01944=86.450,-86.450,14.980,-0.2300,0.2300,0.9400
C01945=91.250,-81.370,14.980,-0.2500,0.2200,0.9400
C01946=95.360,-76.530,14.980,-0.2600,0.2100,0.9400
C01947=98.880,-72.090,15.000,-0.2500,0.2000,0.9500
